RoboDK station: PROYECTO DE MECANIZADO Resuelto.rdk

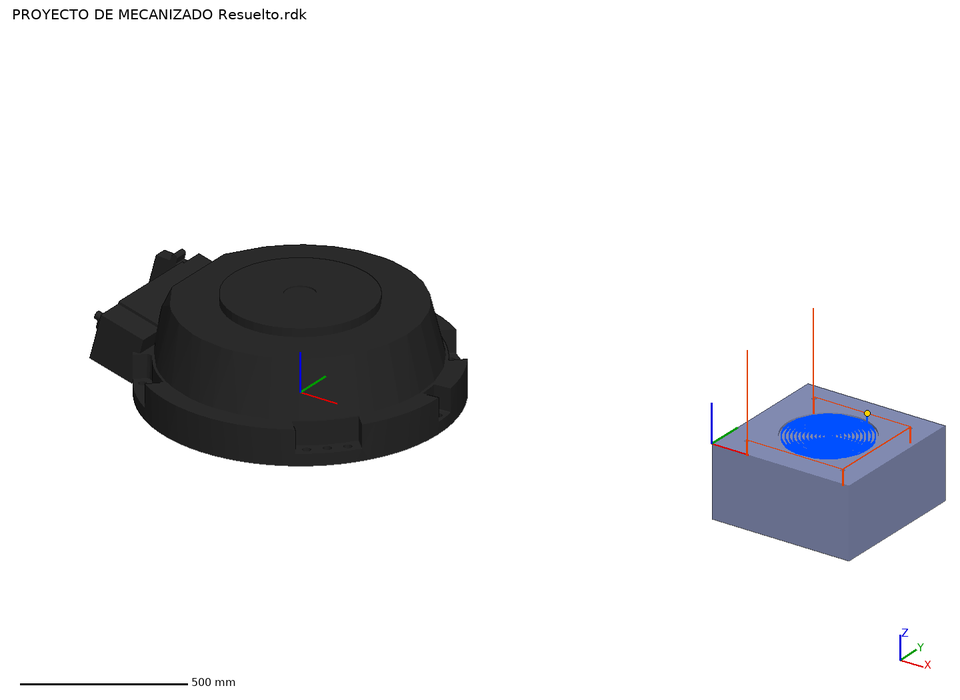
[picture v0: the station drawn from its stored meshes, robots at their saved joint values, targets as dots, program paths as lines]
Station PROYECTO DE MECANIZADO Resuelto (saved by RoboDK 5.7.5). Poses are relative to the parent item; angles as X-Y-Z fixed-axis rotations.
  - frame ORIGEN at (0, 0, 0) mm
  - frame KUKA KR 200 comp Base at (0, 0, 0) mm
    - robot KUKA KR 200 comp: 6 axes
        joint limits [-185, -142, -120, -350, -120, -350] to [185, 0, 148, 350, 120, 350]; home [0, -90, 90, 0, 0, 0]; saved at [-18.305, -63.639, 118.623, 158.005, 56.991, -167.59]
      - tool Teknomotor ATC710039 Spindle, TCP at (296, 0, 80.3) mm, rotated rx 0 ry 90 rz 0 deg, size 475 x 150 x 192.7 mm
        - object ENDMILL_D16_150 at (0, 0, 0) mm, rotated rx 180 ry 0 rz 0 deg, size 16 x 16 x 150 mm, geometry from ENDMILL_D16_150.IGS
  - frame MECANIZADO at (1500, 0, 250) mm
    - object 500x500x250 at (0, 0, 0) mm, size 500 x 500 x 250 mm, geometry from 500x500x250.STEP
  - machining project Machining1 settings: C:/Users/Escritorio/Desktop/pocket_circular (2).gcode | rotZ(0) | rotX(0)*rotY(0)
  - program Machining1 (4843 instructions, listed below)
  - machining project Machining2 settings: C:/Users/Escritorio/Documents/Repos/Proyecto_Tec_12/Proyecto Mecanizado/PROGRAMACION_MANUAL.gcode | rotZ(0) | rotX(0)*rotY(0) | rotz(0) | onStart | onPathStart | onApproach | onPoint | onRetract | onFinish | SetRPM(%1) | SetTool(%1) | Extruder(%1) | default | default | OutOnMov(%1) | OutOffMov(%1) | onPathFinish | M_RunCode(%1)
  - program Machining2 (40 instructions, listed below)
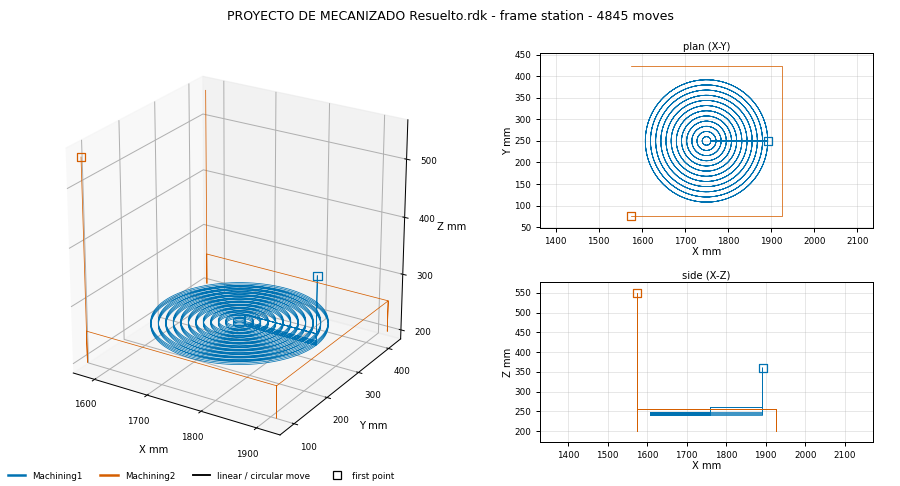
[picture p0: tool path of PROYECTO DE MECANIZADO Resuelto.rdk in frame station, 4845 of 4845 moves have a stored position in this frame; points joined in program order, loops and branches not executed]

--- program Machining1 (robot KUKA KR 200 comp) ---
  Suave(1)
  Establecer velocidad (1000.0 mm/s)
  Est. Ref.: MECANIZADO
  Est. herr: Teknomotor ATC710039 Spindle
  Mostrar Teknomotor ATC710039 Spindle
  MoveJ 1 to (392, 250, 110) mm, rotated rx 180 ry 0 rz -180 deg; joints [-8.871, -45.644, 100.623, 169.209, 55.458, -173.832]
  MoveL 2 to (392, 250, 110) mm, rotated rx 180 ry 0 rz -180 deg; joints [-8.871, -45.644, 100.623, 169.209, 55.458, -173.832]
  MoveL 3 to (392, 250, 10) mm, rotated rx -180 ry 0 rz -180 deg; joints [-8.871, -40.818, 99.818, 169.68, 59.411, -174.706]
  MoveL 4 to (392, 250, 10) mm, rotated rx -180 ry 0 rz -180 deg; joints [-8.871, -40.818, 99.818, 169.68, 59.411, -174.706]
  Establecer velocidad (1000.0 mm/s)
  MoveL 5 to (392, 250, 10) mm, rotated rx -180 ry 0 rz -180 deg; joints [-8.871, -40.818, 99.818, 169.68, 59.411, -174.706]
  Establecer velocidad (1.7 mm/s)
  MoveL 6 to (392, 250, -2.5) mm, rotated rx 180 ry 0 rz 180 deg; joints [-8.871, -40.203, 99.678, 169.73, 59.879, -174.804]
  Establecer velocidad (16.7 mm/s)
  MoveL 7 to (392, 250, -2.5) mm, rotated rx 180 ry 0 rz 180 deg; joints [-8.871, -40.203, 99.678, 169.73, 59.879, -174.804]
  MoveL 8 to (391.71, 259.01, -2.5) mm, rotated rx -180 ry 0 rz -180 deg; joints [-9.187, -40.173, 99.598, 169.361, 59.858, -174.611]
  MoveL 9 to (390.86, 267.98, -2.5) mm, rotated rx -180 ry 0 rz -180 deg; joints [-9.505, -40.157, 99.555, 168.992, 59.862, -174.422]
  MoveL 10 to (389.43, 276.87, -2.5) mm, rotated rx 180 ry 0 rz 180 deg; joints [-9.823, -40.155, 99.548, 168.626, 59.889, -174.237]
  MoveL 11 to (387.45, 285.66, -2.5) mm, rotated rx 180 ry 0 rz 180 deg; joints [-10.141, -40.166, 99.579, 168.263, 59.941, -174.059]
  MoveL 12 to (384.91, 294.31, -2.5) mm, rotated rx 180 ry 0 rz 180 deg; joints [-10.457, -40.191, 99.647, 167.904, 60.016, -173.887]
  MoveL 13 to (381.83, 302.78, -2.5) mm, rotated rx 180 ry 0 rz 180 deg; joints [-10.771, -40.229, 99.751, 167.552, 60.114, -173.723]
  MoveL 14 to (378.22, 311.03, -2.5) mm, rotated rx 180 ry 0 rz -180 deg; joints [-11.082, -40.281, 99.891, 167.207, 60.235, -173.568]
  MoveL 15 to (374.09, 319.04, -2.5) mm, rotated rx -180 ry 0 rz -180 deg; joints [-11.389, -40.346, 100.067, 166.87, 60.378, -173.423]
  MoveL 16 to (369.46, 326.77, -2.5) mm, rotated rx -180 ry 0 rz -180 deg; joints [-11.691, -40.424, 100.278, 166.543, 60.543, -173.289]
  MoveL 17 to (364.35, 334.19, -2.5) mm, rotated rx 180 ry 0 rz 180 deg; joints [-11.987, -40.513, 100.524, 166.226, 60.729, -173.165]
  MoveL 18 to (358.78, 341.28, -2.5) mm, rotated rx -180 ry 0 rz -180 deg; joints [-12.275, -40.615, 100.802, 165.922, 60.935, -173.054]
  MoveL 19 to (352.77, 347.99, -2.5) mm, rotated rx 180 ry 0 rz 180 deg; joints [-12.556, -40.729, 101.113, 165.631, 61.161, -172.955]
  MoveL 20 to (346.35, 354.31, -2.5) mm, rotated rx -180 ry 0 rz 180 deg; joints [-12.828, -40.853, 101.455, 165.353, 61.405, -172.87]
  MoveL 21 to (339.54, 360.21, -2.5) mm, rotated rx -180 ry 0 rz 180 deg; joints [-13.089, -40.987, 101.826, 165.091, 61.667, -172.798]
  MoveL 22 to (332.37, 365.67, -2.5) mm, rotated rx 180 ry 0 rz 180 deg; joints [-13.34, -41.131, 102.226, 164.844, 61.945, -172.74]
  MoveL 23 to (324.87, 370.66, -2.5) mm, rotated rx 180 ry 0 rz 180 deg; joints [-13.579, -41.284, 102.653, 164.614, 62.239, -172.696]
  MoveL 24 to (317.06, 375.17, -2.5) mm, rotated rx -180 ry 0 rz 180 deg; joints [-13.806, -41.445, 103.104, 164.401, 62.548, -172.666]
  MoveL 25 to (308.99, 379.17, -2.5) mm, rotated rx 180 ry 0 rz 180 deg; joints [-14.018, -41.614, 103.579, 164.206, 62.87, -172.65]
  MoveL 26 to (300.68, 382.65, -2.5) mm, rotated rx 180 ry 0 rz -180 deg; joints [-14.217, -41.789, 104.076, 164.03, 63.204, -172.649]
  MoveL 27 to (292.16, 385.6, -2.5) mm, rotated rx 180 ry 0 rz 180 deg; joints [-14.399, -41.97, 104.592, 163.874, 63.55, -172.662]
  MoveL 28 to (283.48, 388, -2.5) mm, rotated rx -180 ry 0 rz 180 deg; joints [-14.566, -42.156, 105.126, 163.737, 63.905, -172.688]
  MoveL 29 to (274.66, 389.84, -2.5) mm, rotated rx 180 ry 0 rz -180 deg; joints [-14.715, -42.347, 105.675, 163.622, 64.269, -172.728]
  MoveL 30 to (265.74, 391.13, -2.5) mm, rotated rx 180 ry 0 rz 180 deg; joints [-14.847, -42.54, 106.238, 163.527, 64.64, -172.782]
  MoveL 31 to (256.76, 391.84, -2.5) mm, rotated rx -180 ry 0 rz 180 deg; joints [-14.96, -42.736, 106.813, 163.454, 65.017, -172.848]
  MoveL 32 to (247.75, 391.98, -2.5) mm, rotated rx -180 ry 0 rz -180 deg; joints [-15.054, -42.934, 107.397, 163.402, 65.399, -172.927]
  MoveL 33 to (238.75, 391.55, -2.5) mm, rotated rx -180 ry 0 rz -180 deg; joints [-15.127, -43.132, 107.987, 163.373, 65.784, -173.017]
  MoveL 34 to (229.79, 390.55, -2.5) mm, rotated rx -180 ry 0 rz -180 deg; joints [-15.18, -43.33, 108.583, 163.367, 66.171, -173.118]
  MoveL 35 to (220.92, 388.99, -2.5) mm, rotated rx -180 ry 0 rz -180 deg; joints [-15.211, -43.526, 109.18, 163.383, 66.559, -173.229]
  MoveL 36 to (212.16, 386.87, -2.5) mm, rotated rx -180 ry 0 rz 180 deg; joints [-15.221, -43.721, 109.778, 163.422, 66.946, -173.351]
  MoveL 37 to (203.56, 384.19, -2.5) mm, rotated rx 180 ry 0 rz -180 deg; joints [-15.208, -43.914, 110.373, 163.484, 67.331, -173.48]
  MoveL 38 to (195.14, 380.97, -2.5) mm, rotated rx 180 ry 0 rz 180 deg; joints [-15.173, -44.102, 110.964, 163.569, 67.712, -173.618]
  MoveL 39 to (186.94, 377.23, -2.5) mm, rotated rx -180 ry 0 rz -180 deg; joints [-15.115, -44.287, 111.547, 163.677, 68.088, -173.763]
  MoveL 40 to (179, 372.98, -2.5) mm, rotated rx -180 ry 0 rz 180 deg; joints [-15.034, -44.466, 112.121, 163.808, 68.458, -173.914]
  MoveL 41 to (171.34, 368.22, -2.5) mm, rotated rx 180 ry 0 rz 180 deg; joints [-14.929, -44.64, 112.683, 163.961, 68.82, -174.07]
  MoveL 42 to (164, 363, -2.5) mm, rotated rx 180 ry 0 rz -180 deg; joints [-14.802, -44.808, 113.231, 164.137, 69.173, -174.231]
  MoveL 43 to (157.01, 357.32, -2.5) mm, rotated rx 180 ry 0 rz -180 deg; joints [-14.652, -44.969, 113.762, 164.335, 69.514, -174.395]
  MoveL 44 to (150.39, 351.2, -2.5) mm, rotated rx 180 ry 0 rz 180 deg; joints [-14.479, -45.122, 114.275, 164.554, 69.844, -174.561]
  MoveL 45 to (144.17, 344.68, -2.5) mm, rotated rx -180 ry 0 rz 180 deg; joints [-14.283, -45.268, 114.767, 164.794, 70.16, -174.729]
  MoveL 46 to (138.38, 337.78, -2.5) mm, rotated rx -180 ry 0 rz 180 deg; joints [-14.067, -45.405, 115.236, 165.054, 70.46, -174.898]
  MoveL 47 to (133.04, 330.52, -2.5) mm, rotated rx 180 ry 0 rz 180 deg; joints [-13.829, -45.533, 115.679, 165.334, 70.744, -175.067]
  MoveL 48 to (128.17, 322.94, -2.5) mm, rotated rx 180 ry 0 rz 180 deg; joints [-13.571, -45.653, 116.096, 165.632, 71.01, -175.235]
  MoveL 49 to (123.79, 315.07, -2.5) mm, rotated rx 180 ry 0 rz -180 deg; joints [-13.294, -45.763, 116.484, 165.947, 71.257, -175.402]
  MoveL 50 to (119.91, 306.93, -2.5) mm, rotated rx -180 ry 0 rz -180 deg; joints [-12.999, -45.863, 116.841, 166.278, 71.484, -175.566]
  MoveL 51 to (116.56, 298.57, -2.5) mm, rotated rx -180 ry 0 rz -180 deg; joints [-12.687, -45.953, 117.166, 166.624, 71.688, -175.727]
  MoveL 52 to (113.75, 290.01, -2.5) mm, rotated rx 180 ry 0 rz 180 deg; joints [-12.36, -46.034, 117.458, 166.983, 71.87, -175.885]
  MoveL 53 to (111.49, 281.28, -2.5) mm, rotated rx 180 ry 0 rz -180 deg; joints [-12.019, -46.104, 117.714, 167.355, 72.027, -176.04]
  MoveL 54 to (109.78, 272.44, -2.5) mm, rotated rx -180 ry 0 rz 180 deg; joints [-11.666, -46.164, 117.934, 167.736, 72.16, -176.19]
  MoveL 55 to (108.64, 263.5, -2.5) mm, rotated rx 180 ry 0 rz -180 deg; joints [-11.303, -46.213, 118.117, 168.125, 72.267, -176.335]
  MoveL 56 to (108.07, 254.51, -2.5) mm, rotated rx -180 ry 0 rz 180 deg; joints [-10.931, -46.252, 118.261, 168.522, 72.347, -176.476]
  MoveL 57 to (108.07, 245.49, -2.5) mm, rotated rx 180 ry 0 rz -180 deg; joints [-10.553, -46.28, 118.367, 168.922, 72.4, -176.612]
  MoveL 58 to (108.64, 236.5, -2.5) mm, rotated rx 180 ry 0 rz -180 deg; joints [-10.17, -46.298, 118.434, 169.326, 72.426, -176.743]
  MoveL 59 to (109.78, 227.56, -2.5) mm, rotated rx -180 ry 0 rz 180 deg; joints [-9.785, -46.305, 118.46, 169.731, 72.423, -176.868]
  MoveL 60 to (111.49, 218.72, -2.5) mm, rotated rx -180 ry 0 rz -180 deg; joints [-9.4, -46.302, 118.447, 170.134, 72.393, -176.989]
  MoveL 61 to (113.75, 209.99, -2.5) mm, rotated rx -180 ry 0 rz -180 deg; joints [-9.016, -46.288, 118.395, 170.534, 72.335, -177.104]
  MoveL 62 to (116.56, 201.43, -2.5) mm, rotated rx 180 ry 0 rz -180 deg; joints [-8.636, -46.263, 118.302, 170.929, 72.25, -177.213]
  MoveL 63 to (119.91, 193.07, -2.5) mm, rotated rx -180 ry 0 rz 180 deg; joints [-8.262, -46.228, 118.171, 171.316, 72.137, -177.318]
  MoveL 64 to (123.79, 184.93, -2.5) mm, rotated rx 180 ry 0 rz -180 deg; joints [-7.896, -46.182, 118.001, 171.695, 71.998, -177.417]
  MoveL 65 to (128.17, 177.06, -2.5) mm, rotated rx -180 ry 0 rz 180 deg; joints [-7.539, -46.126, 117.794, 172.063, 71.832, -177.511]
  MoveL 66 to (133.04, 169.48, -2.5) mm, rotated rx 180 ry 0 rz 180 deg; joints [-7.194, -46.059, 117.55, 172.418, 71.642, -177.599]
  MoveL 67 to (138.38, 162.22, -2.5) mm, rotated rx 180 ry 0 rz -180 deg; joints [-6.862, -45.982, 117.271, 172.759, 71.427, -177.683]
  MoveL 68 to (144.17, 155.32, -2.5) mm, rotated rx -180 ry 0 rz -180 deg; joints [-6.544, -45.895, 116.957, 173.085, 71.19, -177.76]
  MoveL 69 to (150.39, 148.8, -2.5) mm, rotated rx 180 ry 0 rz -180 deg; joints [-6.243, -45.799, 116.611, 173.392, 70.931, -177.833]
  MoveL 70 to (157.01, 142.68, -2.5) mm, rotated rx 180 ry 0 rz -180 deg; joints [-5.96, -45.692, 116.233, 173.682, 70.651, -177.899]
  MoveL 71 to (164, 137, -2.5) mm, rotated rx -180 ry 0 rz 180 deg; joints [-5.695, -45.576, 115.826, 173.951, 70.352, -177.959]
  MoveL 72 to (171.34, 131.78, -2.5) mm, rotated rx 180 ry 0 rz -180 deg; joints [-5.45, -45.45, 115.392, 174.2, 70.036, -178.014]
  MoveL 73 to (179, 127.02, -2.5) mm, rotated rx 180 ry 0 rz 180 deg; joints [-5.226, -45.316, 114.931, 174.427, 69.704, -178.061]
  MoveL 74 to (186.94, 122.77, -2.5) mm, rotated rx -180 ry 0 rz 180 deg; joints [-5.024, -45.174, 114.447, 174.631, 69.357, -178.102]
  MoveL 75 to (195.14, 119.03, -2.5) mm, rotated rx 180 ry 0 rz 180 deg; joints [-4.843, -45.023, 113.941, 174.812, 68.997, -178.136]
  MoveL 76 to (203.56, 115.81, -2.5) mm, rotated rx 180 ry 0 rz 180 deg; joints [-4.685, -44.864, 113.416, 174.969, 68.627, -178.162]
  MoveL 77 to (212.16, 113.13, -2.5) mm, rotated rx 180 ry 0 rz -180 deg; joints [-4.549, -44.699, 112.874, 175.101, 68.247, -178.181]
  MoveL 78 to (220.92, 111.01, -2.5) mm, rotated rx -180 ry 0 rz 180 deg; joints [-4.437, -44.527, 112.316, 175.209, 67.859, -178.191]
  MoveL 79 to (229.79, 109.45, -2.5) mm, rotated rx -180 ry 0 rz -180 deg; joints [-4.348, -44.349, 111.746, 175.292, 67.466, -178.192]
  MoveL 80 to (238.75, 108.45, -2.5) mm, rotated rx -180 ry 0 rz 180 deg; joints [-4.282, -44.167, 111.166, 175.35, 67.067, -178.185]
  MoveL 81 to (247.75, 108.02, -2.5) mm, rotated rx -180 ry 0 rz -180 deg; joints [-4.239, -43.979, 110.578, 175.383, 66.666, -178.168]
  MoveL 82 to (256.76, 108.16, -2.5) mm, rotated rx -180 ry 0 rz -180 deg; joints [-4.218, -43.788, 109.984, 175.391, 66.264, -178.141]
  MoveL 83 to (265.74, 108.87, -2.5) mm, rotated rx 180 ry 0 rz 180 deg; joints [-4.22, -43.594, 109.387, 175.375, 65.863, -178.105]
  MoveL 84 to (274.66, 110.16, -2.5) mm, rotated rx 180 ry 0 rz 180 deg; joints [-4.244, -43.398, 108.789, 175.334, 65.463, -178.059]
  MoveL 85 to (283.48, 112, -2.5) mm, rotated rx 180 ry 0 rz 180 deg; joints [-4.29, -43.2, 108.193, 175.268, 65.067, -178.002]
  MoveL 86 to (292.16, 114.4, -2.5) mm, rotated rx -180 ry 0 rz 180 deg; joints [-4.356, -43.002, 107.6, 175.18, 64.677, -177.934]
  MoveL 87 to (300.68, 117.35, -2.5) mm, rotated rx -180 ry 0 rz -180 deg; joints [-4.443, -42.804, 107.014, 175.068, 64.293, -177.856]
  MoveL 88 to (308.99, 120.83, -2.5) mm, rotated rx 180 ry 0 rz 180 deg; joints [-4.549, -42.608, 106.436, 174.934, 63.917, -177.768]
  MoveL 89 to (317.06, 124.83, -2.5) mm, rotated rx -180 ry 0 rz -180 deg; joints [-4.674, -42.413, 105.868, 174.778, 63.55, -177.669]
  MoveL 90 to (324.87, 129.34, -2.5) mm, rotated rx -180 ry 0 rz -180 deg; joints [-4.818, -42.222, 105.314, 174.601, 63.195, -177.559]
  MoveL 91 to (332.37, 134.33, -2.5) mm, rotated rx -180 ry 0 rz 180 deg; joints [-4.978, -42.034, 104.774, 174.403, 62.852, -177.44]
  MoveL 92 to (339.54, 139.79, -2.5) mm, rotated rx -180 ry 0 rz -180 deg; joints [-5.156, -41.851, 104.252, 174.186, 62.522, -177.31]
  MoveL 93 to (346.35, 145.69, -2.5) mm, rotated rx -180 ry 0 rz -180 deg; joints [-5.349, -41.674, 103.748, 173.951, 62.207, -177.171]
  MoveL 94 to (352.77, 152.01, -2.5) mm, rotated rx -180 ry 0 rz 180 deg; joints [-5.557, -41.503, 103.266, 173.698, 61.907, -177.023]
  MoveL 95 to (358.78, 158.72, -2.5) mm, rotated rx -180 ry 0 rz -180 deg; joints [-5.778, -41.339, 102.806, 173.429, 61.625, -176.867]
  MoveL 96 to (364.35, 165.81, -2.5) mm, rotated rx 180 ry 0 rz 180 deg; joints [-6.013, -41.183, 102.37, 173.145, 61.361, -176.702]
  MoveL 97 to (369.46, 173.23, -2.5) mm, rotated rx 180 ry 0 rz 180 deg; joints [-6.26, -41.036, 101.961, 172.846, 61.115, -176.53]
  MoveL 98 to (374.09, 180.96, -2.5) mm, rotated rx 180 ry 0 rz -180 deg; joints [-6.518, -40.898, 101.58, 172.534, 60.89, -176.352]
  MoveL 99 to (378.22, 188.97, -2.5) mm, rotated rx 180 ry 0 rz 180 deg; joints [-6.787, -40.77, 101.228, 172.211, 60.685, -176.168]
  MoveL 100 to (381.83, 197.22, -2.5) mm, rotated rx 180 ry 0 rz 180 deg; joints [-7.064, -40.653, 100.906, 171.877, 60.501, -175.98]
  MoveL 101 to (384.91, 205.69, -2.5) mm, rotated rx 180 ry 0 rz 180 deg; joints [-7.35, -40.547, 100.616, 171.534, 60.34, -175.787]
  MoveL 102 to (387.45, 214.34, -2.5) mm, rotated rx -180 ry 0 rz 180 deg; joints [-7.643, -40.453, 100.359, 171.183, 60.201, -175.592]
  MoveL 103 to (389.43, 223.13, -2.5) mm, rotated rx 180 ry 0 rz 180 deg; joints [-7.943, -40.371, 100.136, 170.826, 60.085, -175.395]
  MoveL 104 to (390.86, 232.02, -2.5) mm, rotated rx -180 ry 0 rz -180 deg; joints [-8.248, -40.302, 99.948, 170.464, 59.992, -175.198]
  MoveL 105 to (391.71, 240.99, -2.5) mm, rotated rx 180 ry 0 rz 180 deg; joints [-8.558, -40.246, 99.795, 170.098, 59.924, -175]
  MoveL 106 to (392, 250, -2.5) mm, rotated rx 180 ry 0 rz 180 deg; joints [-8.871, -40.203, 99.678, 169.73, 59.879, -174.804]
  MoveL 107 to (380, 250, -2.5) mm, rotated rx -180 ry 0 rz -180 deg; joints [-8.937, -40.511, 100.517, 169.708, 60.406, -174.876]
  MoveL 108 to (379.74, 258.25, -2.5) mm, rotated rx 180 ry 0 rz 180 deg; joints [-9.229, -40.484, 100.443, 169.37, 60.387, -174.701]
  MoveL 109 to (378.95, 266.46, -2.5) mm, rotated rx 180 ry 0 rz -180 deg; joints [-9.521, -40.469, 100.403, 169.032, 60.39, -174.53]
  MoveL 110 to (377.65, 274.6, -2.5) mm, rotated rx 180 ry 0 rz 180 deg; joints [-9.815, -40.467, 100.397, 168.696, 60.415, -174.364]
  MoveL 111 to (375.83, 282.65, -2.5) mm, rotated rx -180 ry 0 rz -180 deg; joints [-10.108, -40.477, 100.425, 168.362, 60.461, -174.202]
  MoveL 112 to (373.51, 290.56, -2.5) mm, rotated rx 180 ry 0 rz -180 deg; joints [-10.4, -40.5, 100.487, 168.033, 60.529, -174.047]
  MoveL 113 to (370.69, 298.32, -2.5) mm, rotated rx -180 ry 0 rz -180 deg; joints [-10.689, -40.535, 100.583, 167.71, 60.619, -173.899]
  MoveL 114 to (367.38, 305.87, -2.5) mm, rotated rx -180 ry 0 rz 180 deg; joints [-10.976, -40.582, 100.712, 167.393, 60.73, -173.759]
  MoveL 115 to (363.6, 313.21, -2.5) mm, rotated rx -180 ry 0 rz -180 deg; joints [-11.259, -40.641, 100.873, 167.083, 60.861, -173.628]
  MoveL 116 to (359.36, 320.28, -2.5) mm, rotated rx 180 ry 0 rz -180 deg; joints [-11.537, -40.712, 101.067, 166.783, 61.012, -173.506]
  MoveL 117 to (354.69, 327.08, -2.5) mm, rotated rx 180 ry 0 rz 180 deg; joints [-11.809, -40.793, 101.291, 166.492, 61.182, -173.395]
  MoveL 118 to (349.59, 333.56, -2.5) mm, rotated rx 180 ry 0 rz -180 deg; joints [-12.075, -40.886, 101.547, 166.212, 61.371, -173.294]
  MoveL 119 to (344.09, 339.71, -2.5) mm, rotated rx -180 ry 0 rz 180 deg; joints [-12.333, -40.989, 101.832, 165.944, 61.578, -173.205]
  MoveL 120 to (338.21, 345.5, -2.5) mm, rotated rx -180 ry 0 rz -180 deg; joints [-12.582, -41.102, 102.145, 165.689, 61.802, -173.127]
  MoveL 121 to (331.97, 350.9, -2.5) mm, rotated rx 180 ry 0 rz 180 deg; joints [-12.823, -41.224, 102.486, 165.448, 62.042, -173.061]
  MoveL 122 to (325.41, 355.89, -2.5) mm, rotated rx 180 ry 0 rz 180 deg; joints [-13.053, -41.355, 102.852, 165.221, 62.298, -173.008]
  MoveL 123 to (318.54, 360.46, -2.5) mm, rotated rx 180 ry 0 rz 180 deg; joints [-13.272, -41.495, 103.243, 165.01, 62.567, -172.967]
  MoveL 124 to (311.4, 364.59, -2.5) mm, rotated rx 180 ry 0 rz 180 deg; joints [-13.479, -41.641, 103.657, 164.814, 62.851, -172.94]
  MoveL 125 to (304, 368.25, -2.5) mm, rotated rx 180 ry 0 rz 180 deg; joints [-13.673, -41.795, 104.092, 164.636, 63.147, -172.925]
  MoveL 126 to (296.4, 371.44, -2.5) mm, rotated rx -180 ry 0 rz 180 deg; joints [-13.854, -41.955, 104.547, 164.474, 63.454, -172.922]
  MoveL 127 to (288.6, 374.14, -2.5) mm, rotated rx 180 ry 0 rz 180 deg; joints [-14.02, -42.12, 105.02, 164.331, 63.771, -172.933]
  MoveL 128 to (280.65, 376.34, -2.5) mm, rotated rx 180 ry 0 rz -180 deg; joints [-14.172, -42.29, 105.51, 164.206, 64.097, -172.956]
  MoveL 129 to (272.57, 378.03, -2.5) mm, rotated rx 180 ry 0 rz -180 deg; joints [-14.307, -42.463, 106.013, 164.101, 64.431, -172.991]
  MoveL 130 to (264.41, 379.2, -2.5) mm, rotated rx -180 ry 0 rz -180 deg; joints [-14.426, -42.64, 106.53, 164.014, 64.772, -173.039]
  MoveL 131 to (256.19, 379.85, -2.5) mm, rotated rx -180 ry 0 rz 180 deg; joints [-14.527, -42.818, 107.056, 163.948, 65.118, -173.097]
  MoveL 132 to (247.94, 379.98, -2.5) mm, rotated rx 180 ry 0 rz 180 deg; joints [-14.611, -42.999, 107.591, 163.902, 65.469, -173.167]
  MoveL 133 to (239.7, 379.59, -2.5) mm, rotated rx 180 ry 0 rz -180 deg; joints [-14.676, -43.18, 108.132, 163.876, 65.822, -173.248]
  MoveL 134 to (231.5, 378.68, -2.5) mm, rotated rx -180 ry 0 rz 180 deg; joints [-14.722, -43.361, 108.677, 163.872, 66.178, -173.338]
  MoveL 135 to (223.38, 377.24, -2.5) mm, rotated rx 180 ry 0 rz 180 deg; joints [-14.748, -43.541, 109.224, 163.888, 66.534, -173.438]
  MoveL 136 to (215.36, 375.3, -2.5) mm, rotated rx 180 ry 0 rz -180 deg; joints [-14.754, -43.719, 109.771, 163.925, 66.889, -173.547]
  MoveL 137 to (207.48, 372.85, -2.5) mm, rotated rx -180 ry 0 rz 180 deg; joints [-14.74, -43.895, 110.316, 163.983, 67.241, -173.663]
  MoveL 138 to (199.78, 369.91, -2.5) mm, rotated rx 180 ry 0 rz -180 deg; joints [-14.705, -44.068, 110.857, 164.063, 67.591, -173.787]
  MoveL 139 to (192.27, 366.48, -2.5) mm, rotated rx 180 ry 0 rz 180 deg; joints [-14.649, -44.238, 111.391, 164.164, 67.935, -173.918]
  MoveL 140 to (185, 362.58, -2.5) mm, rotated rx 180 ry 0 rz 180 deg; joints [-14.573, -44.402, 111.915, 164.285, 68.274, -174.054]
  MoveL 141 to (177.99, 358.23, -2.5) mm, rotated rx 180 ry 0 rz 180 deg; joints [-14.475, -44.562, 112.429, 164.428, 68.605, -174.195]
  MoveL 142 to (171.27, 353.45, -2.5) mm, rotated rx -180 ry 0 rz 180 deg; joints [-14.356, -44.716, 112.93, 164.59, 68.927, -174.34]
  MoveL 143 to (164.87, 348.25, -2.5) mm, rotated rx 180 ry 0 rz -180 deg; joints [-14.217, -44.864, 113.416, 164.773, 69.239, -174.489]
  MoveL 144 to (158.81, 342.65, -2.5) mm, rotated rx 180 ry 0 rz -180 deg; joints [-14.057, -45.006, 113.885, 164.975, 69.54, -174.64]
  MoveL 145 to (153.12, 336.68, -2.5) mm, rotated rx 180 ry 0 rz 180 deg; joints [-13.877, -45.14, 114.334, 165.196, 69.828, -174.793]
  MoveL 146 to (147.81, 330.36, -2.5) mm, rotated rx -180 ry 0 rz 180 deg; joints [-13.677, -45.266, 114.762, 165.436, 70.102, -174.947]
  MoveL 147 to (142.92, 323.72, -2.5) mm, rotated rx 180 ry 0 rz -180 deg; joints [-13.459, -45.385, 115.167, 165.692, 70.36, -175.101]
  MoveL 148 to (138.46, 316.78, -2.5) mm, rotated rx 180 ry 0 rz 180 deg; joints [-13.223, -45.496, 115.548, 165.966, 70.602, -175.254]
  MoveL 149 to (134.45, 309.57, -2.5) mm, rotated rx -180 ry 0 rz -180 deg; joints [-12.97, -45.597, 115.902, 166.254, 70.827, -175.407]
  MoveL 150 to (130.91, 302.12, -2.5) mm, rotated rx 180 ry 0 rz 180 deg; joints [-12.7, -45.69, 116.228, 166.557, 71.032, -175.558]
  MoveL 151 to (127.84, 294.46, -2.5) mm, rotated rx 180 ry 0 rz 180 deg; joints [-12.416, -45.774, 116.524, 166.874, 71.217, -175.706]
  MoveL 152 to (125.27, 286.63, -2.5) mm, rotated rx -180 ry 0 rz -180 deg; joints [-12.118, -45.849, 116.79, 167.202, 71.382, -175.852]
  MoveL 153 to (123.19, 278.64, -2.5) mm, rotated rx 180 ry 0 rz 180 deg; joints [-11.808, -45.914, 117.024, 167.541, 71.524, -175.995]
  MoveL 154 to (121.63, 270.54, -2.5) mm, rotated rx 180 ry 0 rz 180 deg; joints [-11.487, -45.969, 117.224, 167.888, 71.644, -176.134]
  MoveL 155 to (120.59, 262.36, -2.5) mm, rotated rx 180 ry 0 rz 180 deg; joints [-11.157, -46.015, 117.391, 168.244, 71.74, -176.269]
  MoveL 156 to (120.07, 254.12, -2.5) mm, rotated rx 180 ry 0 rz 180 deg; joints [-10.819, -46.052, 117.522, 168.605, 71.812, -176.4]
  MoveL 157 to (120.07, 245.88, -2.5) mm, rotated rx -180 ry 0 rz -180 deg; joints [-10.476, -46.078, 117.619, 168.97, 71.859, -176.527]
  MoveL 158 to (120.59, 237.64, -2.5) mm, rotated rx -180 ry 0 rz -180 deg; joints [-10.128, -46.094, 117.679, 169.337, 71.882, -176.649]
  MoveL 159 to (121.63, 229.46, -2.5) mm, rotated rx 180 ry 0 rz 180 deg; joints [-9.779, -46.101, 117.704, 169.705, 71.879, -176.767]
  MoveL 160 to (123.19, 221.36, -2.5) mm, rotated rx 180 ry 0 rz 180 deg; joints [-9.429, -46.098, 117.692, 170.072, 71.851, -176.879]
  MoveL 161 to (125.27, 213.37, -2.5) mm, rotated rx 180 ry 0 rz 180 deg; joints [-9.081, -46.085, 117.644, 170.436, 71.798, -176.987]
  MoveL 162 to (127.84, 205.54, -2.5) mm, rotated rx -180 ry 0 rz 180 deg; joints [-8.736, -46.062, 117.56, 170.796, 71.72, -177.09]
  MoveL 163 to (130.91, 197.88, -2.5) mm, rotated rx 180 ry 0 rz 180 deg; joints [-8.396, -46.029, 117.44, 171.149, 71.618, -177.188]
  MoveL 164 to (134.45, 190.43, -2.5) mm, rotated rx 180 ry 0 rz -180 deg; joints [-8.064, -45.986, 117.286, 171.493, 71.491, -177.282]
  MoveL 165 to (138.46, 183.22, -2.5) mm, rotated rx 180 ry 0 rz 180 deg; joints [-7.739, -45.934, 117.097, 171.828, 71.34, -177.37]
  MoveL 166 to (142.92, 176.28, -2.5) mm, rotated rx -180 ry 0 rz 180 deg; joints [-7.425, -45.872, 116.874, 172.152, 71.167, -177.452]
  MoveL 167 to (147.81, 169.64, -2.5) mm, rotated rx 180 ry 0 rz 180 deg; joints [-7.123, -45.801, 116.619, 172.463, 70.972, -177.53]
  MoveL 168 to (153.12, 163.32, -2.5) mm, rotated rx -180 ry 0 rz 180 deg; joints [-6.834, -45.72, 116.333, 172.76, 70.756, -177.602]
  MoveL 169 to (158.81, 157.35, -2.5) mm, rotated rx 180 ry 0 rz 180 deg; joints [-6.559, -45.63, 116.017, 173.041, 70.521, -177.669]
  MoveL 170 to (164.87, 151.75, -2.5) mm, rotated rx 180 ry 0 rz -180 deg; joints [-6.3, -45.532, 115.673, 173.305, 70.266, -177.73]
  MoveL 171 to (171.27, 146.55, -2.5) mm, rotated rx -180 ry 0 rz 180 deg; joints [-6.058, -45.424, 115.301, 173.552, 69.994, -177.786]
  MoveL 172 to (177.99, 141.77, -2.5) mm, rotated rx 180 ry 0 rz -180 deg; joints [-5.833, -45.308, 114.905, 173.779, 69.707, -177.835]
  MoveL 173 to (185, 137.42, -2.5) mm, rotated rx -180 ry 0 rz 180 deg; joints [-5.627, -45.184, 114.484, 173.987, 69.404, -177.878]
  MoveL 174 to (192.27, 133.52, -2.5) mm, rotated rx 180 ry 0 rz -180 deg; joints [-5.44, -45.053, 114.042, 174.175, 69.088, -177.915]
  MoveL 175 to (199.78, 130.09, -2.5) mm, rotated rx 180 ry 0 rz 180 deg; joints [-5.273, -44.914, 113.58, 174.341, 68.761, -177.944]
  MoveL 176 to (207.48, 127.15, -2.5) mm, rotated rx 180 ry 0 rz -180 deg; joints [-5.127, -44.768, 113.1, 174.486, 68.423, -177.967]
  MoveL 177 to (215.36, 124.7, -2.5) mm, rotated rx -180 ry 0 rz 180 deg; joints [-5.001, -44.616, 112.604, 174.608, 68.076, -177.982]
  MoveL 178 to (223.38, 122.76, -2.5) mm, rotated rx -180 ry 0 rz -180 deg; joints [-4.896, -44.458, 112.094, 174.708, 67.722, -177.989]
  MoveL 179 to (231.5, 121.32, -2.5) mm, rotated rx 180 ry 0 rz 180 deg; joints [-4.812, -44.295, 111.573, 174.785, 67.362, -177.988]
  MoveL 180 to (239.7, 120.41, -2.5) mm, rotated rx 180 ry 0 rz 180 deg; joints [-4.749, -44.127, 111.042, 174.84, 66.998, -177.979]
  MoveL 181 to (247.94, 120.02, -2.5) mm, rotated rx 180 ry 0 rz -180 deg; joints [-4.707, -43.955, 110.504, 174.871, 66.632, -177.961]
  MoveL 182 to (256.19, 120.15, -2.5) mm, rotated rx 180 ry 0 rz -180 deg; joints [-4.686, -43.78, 109.96, 174.88, 66.264, -177.935]
  MoveL 183 to (264.41, 120.8, -2.5) mm, rotated rx 180 ry 0 rz 180 deg; joints [-4.685, -43.603, 109.413, 174.867, 65.897, -177.899]
  MoveL 184 to (272.57, 121.98, -2.5) mm, rotated rx -180 ry 0 rz -180 deg; joints [-4.704, -43.423, 108.866, 174.83, 65.531, -177.854]
  MoveL 185 to (280.65, 123.66, -2.5) mm, rotated rx -180 ry 0 rz -180 deg; joints [-4.743, -43.242, 108.32, 174.772, 65.168, -177.8]
  MoveL 186 to (288.6, 125.86, -2.5) mm, rotated rx 180 ry 0 rz 180 deg; joints [-4.802, -43.061, 107.777, 174.692, 64.811, -177.736]
  MoveL 187 to (296.4, 128.56, -2.5) mm, rotated rx -180 ry 0 rz 180 deg; joints [-4.879, -42.881, 107.24, 174.591, 64.459, -177.662]
  MoveL 188 to (304, 131.75, -2.5) mm, rotated rx 180 ry 0 rz -180 deg; joints [-4.974, -42.701, 106.71, 174.469, 64.114, -177.579]
  MoveL 189 to (311.4, 135.41, -2.5) mm, rotated rx 180 ry 0 rz 180 deg; joints [-5.087, -42.524, 106.19, 174.327, 63.778, -177.487]
  MoveL 190 to (318.54, 139.54, -2.5) mm, rotated rx 180 ry 0 rz -180 deg; joints [-5.217, -42.349, 105.682, 174.166, 63.452, -177.385]
  MoveL 191 to (325.41, 144.11, -2.5) mm, rotated rx 180 ry 0 rz -180 deg; joints [-5.363, -42.178, 105.188, 173.986, 63.137, -177.275]
  MoveL 192 to (331.97, 149.1, -2.5) mm, rotated rx -180 ry 0 rz 180 deg; joints [-5.524, -42.011, 104.709, 173.788, 62.835, -177.155]
  MoveL 193 to (338.21, 154.5, -2.5) mm, rotated rx 180 ry 0 rz 180 deg; joints [-5.7, -41.849, 104.247, 173.574, 62.546, -177.027]
  MoveL 194 to (344.09, 160.29, -2.5) mm, rotated rx 180 ry 0 rz -180 deg; joints [-5.89, -41.694, 103.805, 173.343, 62.271, -176.891]
  MoveL 195 to (349.59, 166.44, -2.5) mm, rotated rx 180 ry 0 rz 180 deg; joints [-6.093, -41.544, 103.383, 173.097, 62.012, -176.748]
  MoveL 196 to (354.69, 172.92, -2.5) mm, rotated rx -180 ry 0 rz 180 deg; joints [-6.308, -41.403, 102.984, 172.837, 61.769, -176.598]
  MoveL 197 to (359.36, 179.72, -2.5) mm, rotated rx 180 ry 0 rz -180 deg; joints [-6.534, -41.269, 102.609, 172.563, 61.544, -176.441]
  MoveL 198 to (363.6, 186.79, -2.5) mm, rotated rx -180 ry 0 rz -180 deg; joints [-6.771, -41.143, 102.26, 172.278, 61.337, -176.279]
  MoveL 199 to (367.38, 194.13, -2.5) mm, rotated rx -180 ry 0 rz 180 deg; joints [-7.017, -41.027, 101.937, 171.982, 61.148, -176.111]
  MoveL 200 to (370.69, 201.68, -2.5) mm, rotated rx -180 ry 0 rz 180 deg; joints [-7.273, -40.92, 101.642, 171.676, 60.98, -175.94]
  MoveL 201 to (373.51, 209.44, -2.5) mm, rotated rx 180 ry 0 rz -180 deg; joints [-7.536, -40.824, 101.376, 171.362, 60.831, -175.766]
  MoveL 202 to (375.83, 217.35, -2.5) mm, rotated rx 180 ry 0 rz -180 deg; joints [-7.806, -40.739, 101.141, 171.041, 60.703, -175.589]
  MoveL 203 to (377.65, 225.4, -2.5) mm, rotated rx 180 ry 0 rz -180 deg; joints [-8.082, -40.664, 100.936, 170.713, 60.597, -175.41]
  MoveL 204 to (378.95, 233.54, -2.5) mm, rotated rx 180 ry 0 rz 180 deg; joints [-8.363, -40.601, 100.764, 170.381, 60.511, -175.231]
  MoveL 205 to (379.74, 241.75, -2.5) mm, rotated rx 180 ry 0 rz 180 deg; joints [-8.648, -40.55, 100.624, 170.046, 60.448, -175.053]
  MoveL 206 to (380, 250, -2.5) mm, rotated rx -180 ry 0 rz -180 deg; joints [-8.937, -40.511, 100.517, 169.708, 60.406, -174.876]
  MoveL 207 to (368, 250, -2.5) mm, rotated rx -180 ry 0 rz -180 deg; joints [-9.004, -40.814, 101.349, 169.685, 60.933, -174.947]
  MoveL 208 to (367.76, 257.48, -2.5) mm, rotated rx 180 ry 0 rz -180 deg; joints [-9.27, -40.79, 101.283, 169.377, 60.915, -174.791]
  MoveL 209 to (367.05, 264.94, -2.5) mm, rotated rx -180 ry 0 rz -180 deg; joints [-9.538, -40.777, 101.246, 169.07, 60.917, -174.637]
  MoveL 210 to (365.87, 272.33, -2.5) mm, rotated rx 180 ry 0 rz -180 deg; joints [-9.806, -40.775, 101.241, 168.764, 60.939, -174.488]
  MoveL 211 to (364.22, 279.64, -2.5) mm, rotated rx -180 ry 0 rz -180 deg; joints [-10.075, -40.784, 101.267, 168.461, 60.981, -174.344]
  MoveL 212 to (362.11, 286.82, -2.5) mm, rotated rx -180 ry 0 rz 180 deg; joints [-10.341, -40.805, 101.323, 168.161, 61.043, -174.205]
  MoveL 213 to (359.55, 293.86, -2.5) mm, rotated rx 180 ry 0 rz 180 deg; joints [-10.606, -40.836, 101.41, 167.866, 61.124, -174.072]
  MoveL 214 to (356.55, 300.72, -2.5) mm, rotated rx 180 ry 0 rz 180 deg; joints [-10.868, -40.879, 101.527, 167.578, 61.224, -173.947]
  MoveL 215 to (353.11, 307.37, -2.5) mm, rotated rx -180 ry 0 rz 180 deg; joints [-11.127, -40.932, 101.673, 167.296, 61.343, -173.83]
  MoveL 216 to (349.27, 313.8, -2.5) mm, rotated rx -180 ry 0 rz -180 deg; joints [-11.381, -40.995, 101.849, 167.022, 61.48, -173.721]
  MoveL 217 to (345.02, 319.96, -2.5) mm, rotated rx -180 ry 0 rz -180 deg; joints [-11.629, -41.069, 102.054, 166.757, 61.635, -173.62]
  MoveL 218 to (340.39, 325.85, -2.5) mm, rotated rx -180 ry 0 rz -180 deg; joints [-11.871, -41.153, 102.286, 166.502, 61.807, -173.53]
  MoveL 219 to (335.4, 331.43, -2.5) mm, rotated rx -180 ry 0 rz -180 deg; joints [-12.107, -41.246, 102.545, 166.258, 61.995, -173.45]
  MoveL 220 to (330.06, 336.68, -2.5) mm, rotated rx -180 ry 0 rz -180 deg; joints [-12.334, -41.347, 102.83, 166.026, 62.198, -173.379]
  MoveL 221 to (324.41, 341.59, -2.5) mm, rotated rx -180 ry 0 rz -180 deg; joints [-12.553, -41.458, 103.139, 165.806, 62.417, -173.32]
  MoveL 222 to (318.45, 346.12, -2.5) mm, rotated rx 180 ry 0 rz 180 deg; joints [-12.762, -41.576, 103.472, 165.599, 62.65, -173.272]
  MoveL 223 to (312.21, 350.27, -2.5) mm, rotated rx -180 ry 0 rz 180 deg; joints [-12.961, -41.702, 103.828, 165.407, 62.895, -173.235]
  MoveL 224 to (305.73, 354.01, -2.5) mm, rotated rx -180 ry 0 rz 180 deg; joints [-13.149, -41.834, 104.204, 165.229, 63.153, -173.209]
  MoveL 225 to (299.02, 357.34, -2.5) mm, rotated rx -180 ry 0 rz -180 deg; joints [-13.325, -41.973, 104.6, 165.066, 63.422, -173.195]
  MoveL 226 to (292.11, 360.23, -2.5) mm, rotated rx -180 ry 0 rz -180 deg; joints [-13.488, -42.117, 105.013, 164.92, 63.702, -173.192]
  MoveL 227 to (285.04, 362.68, -2.5) mm, rotated rx 180 ry 0 rz -180 deg; joints [-13.639, -42.266, 105.443, 164.789, 63.991, -173.201]
  MoveL 228 to (277.82, 364.67, -2.5) mm, rotated rx 180 ry 0 rz 180 deg; joints [-13.775, -42.42, 105.888, 164.676, 64.288, -173.22]
  MoveL 229 to (270.49, 366.21, -2.5) mm, rotated rx -180 ry 0 rz 180 deg; joints [-13.896, -42.577, 106.346, 164.581, 64.592, -173.251]
  MoveL 230 to (263.08, 367.27, -2.5) mm, rotated rx -180 ry 0 rz -180 deg; joints [-14.002, -42.737, 106.814, 164.503, 64.903, -173.292]
  MoveL 231 to (255.61, 367.87, -2.5) mm, rotated rx -180 ry 0 rz 180 deg; joints [-14.093, -42.898, 107.293, 164.443, 65.218, -173.344]
  MoveL 232 to (248.13, 367.99, -2.5) mm, rotated rx 180 ry 0 rz -180 deg; joints [-14.167, -43.062, 107.778, 164.402, 65.537, -173.406]
  MoveL 233 to (240.65, 367.63, -2.5) mm, rotated rx -180 ry 0 rz 180 deg; joints [-14.224, -43.226, 108.27, 164.38, 65.859, -173.477]
  MoveL 234 to (233.21, 366.8, -2.5) mm, rotated rx 180 ry 0 rz -180 deg; joints [-14.263, -43.39, 108.765, 164.377, 66.182, -173.557]
  MoveL 235 to (225.83, 365.5, -2.5) mm, rotated rx 180 ry 0 rz 180 deg; joints [-14.284, -43.553, 109.262, 164.393, 66.506, -173.646]
  MoveL 236 to (218.56, 363.73, -2.5) mm, rotated rx -180 ry 0 rz -180 deg; joints [-14.288, -43.715, 109.759, 164.428, 66.829, -173.742]
  MoveL 237 to (211.41, 361.51, -2.5) mm, rotated rx -180 ry 0 rz -180 deg; joints [-14.273, -43.875, 110.253, 164.483, 67.149, -173.846]
  MoveL 238 to (204.41, 358.84, -2.5) mm, rotated rx 180 ry 0 rz -180 deg; joints [-14.239, -44.032, 110.743, 164.556, 67.467, -173.957]
  MoveL 239 to (197.6, 355.73, -2.5) mm, rotated rx -180 ry 0 rz -180 deg; joints [-14.186, -44.186, 111.228, 164.649, 67.78, -174.073]
  MoveL 240 to (191, 352.19, -2.5) mm, rotated rx -180 ry 0 rz -180 deg; joints [-14.114, -44.336, 111.704, 164.761, 68.087, -174.195]
  MoveL 241 to (184.64, 348.24, -2.5) mm, rotated rx 180 ry 0 rz 180 deg; joints [-14.023, -44.482, 112.17, 164.892, 68.387, -174.321]
  MoveL 242 to (178.54, 343.9, -2.5) mm, rotated rx -180 ry 0 rz 180 deg; joints [-13.913, -44.622, 112.624, 165.041, 68.679, -174.452]
  MoveL 243 to (172.73, 339.18, -2.5) mm, rotated rx 180 ry 0 rz 180 deg; joints [-13.785, -44.757, 113.064, 165.209, 68.962, -174.585]
  MoveL 244 to (167.23, 334.1, -2.5) mm, rotated rx 180 ry 0 rz -180 deg; joints [-13.639, -44.886, 113.488, 165.393, 69.234, -174.721]
  MoveL 245 to (162.06, 328.68, -2.5) mm, rotated rx -180 ry 0 rz 180 deg; joints [-13.474, -45.009, 113.895, 165.595, 69.494, -174.859]
  MoveL 246 to (157.25, 322.94, -2.5) mm, rotated rx -180 ry 0 rz -180 deg; joints [-13.292, -45.125, 114.283, 165.813, 69.742, -174.998]
  MoveL 247 to (152.81, 316.91, -2.5) mm, rotated rx 180 ry 0 rz 180 deg; joints [-13.094, -45.233, 114.65, 166.047, 69.975, -175.137]
  MoveL 248 to (148.76, 310.61, -2.5) mm, rotated rx -180 ry 0 rz 180 deg; joints [-12.879, -45.335, 114.994, 166.295, 70.193, -175.276]
  MoveL 249 to (145.12, 304.07, -2.5) mm, rotated rx 180 ry 0 rz -180 deg; joints [-12.65, -45.428, 115.315, 166.558, 70.395, -175.415]
  MoveL 250 to (141.9, 297.31, -2.5) mm, rotated rx -180 ry 0 rz 180 deg; joints [-12.406, -45.513, 115.609, 166.833, 70.58, -175.552]
  MoveL 251 to (139.12, 290.36, -2.5) mm, rotated rx -180 ry 0 rz 180 deg; joints [-12.149, -45.59, 115.878, 167.12, 70.746, -175.688]
  MoveL 252 to (136.78, 283.24, -2.5) mm, rotated rx 180 ry 0 rz 180 deg; joints [-11.879, -45.659, 116.118, 167.417, 70.894, -175.821]
  MoveL 253 to (134.9, 276, -2.5) mm, rotated rx 180 ry 0 rz 180 deg; joints [-11.6, -45.719, 116.329, 167.724, 71.021, -175.952]
  MoveL 254 to (133.48, 268.64, -2.5) mm, rotated rx 180 ry 0 rz 180 deg; joints [-11.31, -45.77, 116.511, 168.038, 71.129, -176.08]
  MoveL 255 to (132.53, 261.22, -2.5) mm, rotated rx 180 ry 0 rz 180 deg; joints [-11.013, -45.813, 116.661, 168.359, 71.214, -176.204]
  MoveL 256 to (132.06, 253.74, -2.5) mm, rotated rx -180 ry 0 rz -180 deg; joints [-10.709, -45.846, 116.78, 168.685, 71.279, -176.325]
  MoveL 257 to (132.06, 246.26, -2.5) mm, rotated rx -180 ry 0 rz -180 deg; joints [-10.4, -45.87, 116.867, 169.015, 71.321, -176.443]
  MoveL 258 to (132.53, 238.78, -2.5) mm, rotated rx -180 ry 0 rz 180 deg; joints [-10.087, -45.886, 116.922, 169.347, 71.34, -176.556]
  MoveL 259 to (133.48, 231.36, -2.5) mm, rotated rx 180 ry 0 rz 180 deg; joints [-9.773, -45.892, 116.944, 169.679, 71.337, -176.665]
  MoveL 260 to (134.9, 224, -2.5) mm, rotated rx 180 ry 0 rz -180 deg; joints [-9.458, -45.889, 116.933, 170.01, 71.312, -176.77]
  MoveL 261 to (136.78, 216.76, -2.5) mm, rotated rx -180 ry 0 rz 180 deg; joints [-9.145, -45.877, 116.89, 170.338, 71.264, -176.87]
  MoveL 262 to (139.12, 209.64, -2.5) mm, rotated rx -180 ry 0 rz 180 deg; joints [-8.835, -45.855, 116.814, 170.663, 71.193, -176.966]
  MoveL 263 to (141.9, 202.69, -2.5) mm, rotated rx -180 ry 0 rz -180 deg; joints [-8.529, -45.825, 116.706, 170.981, 71.1, -177.057]
  MoveL 264 to (145.12, 195.93, -2.5) mm, rotated rx 180 ry 0 rz -180 deg; joints [-8.229, -45.786, 116.566, 171.293, 70.986, -177.143]
  MoveL 265 to (148.76, 189.39, -2.5) mm, rotated rx -180 ry 0 rz -180 deg; joints [-7.937, -45.738, 116.395, 171.595, 70.85, -177.225]
  MoveL 266 to (152.81, 183.09, -2.5) mm, rotated rx 180 ry 0 rz -180 deg; joints [-7.653, -45.681, 116.194, 171.888, 70.694, -177.302]
  MoveL 267 to (157.25, 177.06, -2.5) mm, rotated rx 180 ry 0 rz 180 deg; joints [-7.38, -45.615, 115.964, 172.169, 70.518, -177.374]
  MoveL 268 to (162.06, 171.32, -2.5) mm, rotated rx -180 ry 0 rz 180 deg; joints [-7.119, -45.541, 115.705, 172.437, 70.323, -177.44]
  MoveL 269 to (167.23, 165.9, -2.5) mm, rotated rx 180 ry 0 rz 180 deg; joints [-6.87, -45.458, 115.419, 172.692, 70.111, -177.502]
  MoveL 270 to (172.73, 160.82, -2.5) mm, rotated rx 180 ry 0 rz -180 deg; joints [-6.636, -45.368, 115.108, 172.931, 69.881, -177.558]
  MoveL 271 to (178.54, 156.1, -2.5) mm, rotated rx -180 ry 0 rz -180 deg; joints [-6.416, -45.269, 114.771, 173.155, 69.636, -177.608]
  MoveL 272 to (184.64, 151.76, -2.5) mm, rotated rx 180 ry 0 rz 180 deg; joints [-6.212, -45.163, 114.412, 173.361, 69.376, -177.652]
  MoveL 273 to (191, 147.81, -2.5) mm, rotated rx -180 ry 0 rz 180 deg; joints [-6.024, -45.05, 114.031, 173.55, 69.103, -177.691]
  MoveL 274 to (197.6, 144.27, -2.5) mm, rotated rx 180 ry 0 rz 180 deg; joints [-5.853, -44.929, 113.631, 173.721, 68.818, -177.723]
  MoveL 275 to (204.41, 141.16, -2.5) mm, rotated rx 180 ry 0 rz -180 deg; joints [-5.701, -44.802, 113.212, 173.872, 68.522, -177.749]
  MoveL 276 to (211.41, 138.49, -2.5) mm, rotated rx -180 ry 0 rz -180 deg; joints [-5.566, -44.669, 112.777, 174.004, 68.216, -177.768]
  MoveL 277 to (218.56, 136.27, -2.5) mm, rotated rx 180 ry 0 rz 180 deg; joints [-5.45, -44.531, 112.328, 174.117, 67.903, -177.78]
  MoveL 278 to (225.83, 134.5, -2.5) mm, rotated rx -180 ry 0 rz 180 deg; joints [-5.353, -44.387, 111.866, 174.208, 67.582, -177.785]
  MoveL 279 to (233.21, 133.2, -2.5) mm, rotated rx -180 ry 0 rz 180 deg; joints [-5.274, -44.238, 111.393, 174.28, 67.257, -177.782]
  MoveL 280 to (240.65, 132.37, -2.5) mm, rotated rx 180 ry 0 rz 180 deg; joints [-5.215, -44.086, 110.911, 174.33, 66.927, -177.772]
  MoveL 281 to (248.13, 132.01, -2.5) mm, rotated rx -180 ry 0 rz 180 deg; joints [-5.174, -43.93, 110.423, 174.36, 66.595, -177.754]
  MoveL 282 to (255.61, 132.13, -2.5) mm, rotated rx 180 ry 0 rz 180 deg; joints [-5.153, -43.771, 109.93, 174.37, 66.261, -177.727]
  MoveL 283 to (263.08, 132.73, -2.5) mm, rotated rx 180 ry 0 rz 180 deg; joints [-5.15, -43.609, 109.433, 174.358, 65.928, -177.693]
  MoveL 284 to (270.49, 133.79, -2.5) mm, rotated rx 180 ry 0 rz 180 deg; joints [-5.165, -43.446, 108.936, 174.327, 65.596, -177.65]
  MoveL 285 to (277.82, 135.33, -2.5) mm, rotated rx -180 ry 0 rz -180 deg; joints [-5.198, -43.282, 108.44, 174.275, 65.267, -177.598]
  MoveL 286 to (285.04, 137.32, -2.5) mm, rotated rx 180 ry 0 rz -180 deg; joints [-5.249, -43.118, 107.948, 174.204, 64.942, -177.538]
  MoveL 287 to (292.11, 139.77, -2.5) mm, rotated rx -180 ry 0 rz -180 deg; joints [-5.317, -42.955, 107.46, 174.113, 64.622, -177.47]
  MoveL 288 to (299.02, 142.66, -2.5) mm, rotated rx -180 ry 0 rz -180 deg; joints [-5.402, -42.792, 106.979, 174.004, 64.309, -177.393]
  MoveL 289 to (305.73, 145.99, -2.5) mm, rotated rx -180 ry 0 rz -180 deg; joints [-5.503, -42.632, 106.506, 173.876, 64.004, -177.307]
  MoveL 290 to (312.21, 149.73, -2.5) mm, rotated rx -180 ry 0 rz -180 deg; joints [-5.619, -42.474, 106.045, 173.73, 63.708, -177.214]
  MoveL 291 to (318.45, 153.88, -2.5) mm, rotated rx 180 ry 0 rz 180 deg; joints [-5.75, -42.319, 105.595, 173.568, 63.421, -177.112]
  MoveL 292 to (324.41, 158.41, -2.5) mm, rotated rx 180 ry 0 rz 180 deg; joints [-5.896, -42.168, 105.16, 173.389, 63.146, -177.003]
  MoveL 293 to (330.06, 163.32, -2.5) mm, rotated rx 180 ry 0 rz -180 deg; joints [-6.055, -42.022, 104.741, 173.194, 62.883, -176.886]
  MoveL 294 to (335.4, 168.57, -2.5) mm, rotated rx 180 ry 0 rz 180 deg; joints [-6.226, -41.882, 104.338, 172.985, 62.633, -176.763]
  MoveL 295 to (340.39, 174.15, -2.5) mm, rotated rx -180 ry 0 rz -180 deg; joints [-6.41, -41.747, 103.955, 172.762, 62.397, -176.632]
  MoveL 296 to (345.02, 180.04, -2.5) mm, rotated rx 180 ry 0 rz -180 deg; joints [-6.605, -41.619, 103.593, 172.526, 62.176, -176.496]
  MoveL 297 to (349.27, 186.2, -2.5) mm, rotated rx 180 ry 0 rz 180 deg; joints [-6.811, -41.498, 103.252, 172.279, 61.971, -176.354]
  MoveL 298 to (353.11, 192.63, -2.5) mm, rotated rx -180 ry 0 rz -180 deg; joints [-7.027, -41.385, 102.934, 172.02, 61.782, -176.208]
  MoveL 299 to (356.55, 199.28, -2.5) mm, rotated rx 180 ry 0 rz -180 deg; joints [-7.251, -41.28, 102.64, 171.751, 61.611, -176.057]
  MoveL 300 to (359.55, 206.14, -2.5) mm, rotated rx -180 ry 0 rz 180 deg; joints [-7.484, -41.184, 102.372, 171.474, 61.457, -175.903]
  MoveL 301 to (362.11, 213.18, -2.5) mm, rotated rx -180 ry 0 rz 180 deg; joints [-7.724, -41.097, 102.131, 171.188, 61.321, -175.745]
  MoveL 302 to (364.22, 220.36, -2.5) mm, rotated rx -180 ry 0 rz 180 deg; joints [-7.97, -41.02, 101.917, 170.896, 61.205, -175.586]
  MoveL 303 to (365.87, 227.67, -2.5) mm, rotated rx -180 ry 0 rz -180 deg; joints [-8.222, -40.953, 101.731, 170.599, 61.107, -175.426]
  MoveL 304 to (367.05, 235.06, -2.5) mm, rotated rx 180 ry 0 rz 180 deg; joints [-8.479, -40.896, 101.574, 170.297, 61.029, -175.266]
  MoveL 305 to (367.76, 242.52, -2.5) mm, rotated rx 180 ry 0 rz -180 deg; joints [-8.74, -40.85, 101.447, 169.992, 60.971, -175.106]
  MoveL 306 to (368, 250, -2.5) mm, rotated rx -180 ry 0 rz -180 deg; joints [-9.004, -40.814, 101.349, 169.685, 60.933, -174.947]
  MoveL 307 to (356, 250, -2.5) mm, rotated rx 180 ry 0 rz 180 deg; joints [-9.072, -41.114, 102.177, 169.66, 61.459, -175.018]
  MoveL 308 to (355.79, 256.72, -2.5) mm, rotated rx -180 ry 0 rz -180 deg; joints [-9.313, -41.092, 102.117, 169.383, 61.443, -174.879]
  MoveL 309 to (355.15, 263.42, -2.5) mm, rotated rx 180 ry 0 rz -180 deg; joints [-9.555, -41.08, 102.085, 169.106, 61.444, -174.744]
  MoveL 310 to (354.08, 270.06, -2.5) mm, rotated rx -180 ry 0 rz 180 deg; joints [-9.798, -41.078, 102.08, 168.831, 61.464, -174.611]
  MoveL 311 to (352.6, 276.62, -2.5) mm, rotated rx -180 ry 0 rz -180 deg; joints [-10.041, -41.087, 102.103, 168.557, 61.501, -174.484]
  MoveL 312 to (350.71, 283.08, -2.5) mm, rotated rx -180 ry 0 rz 180 deg; joints [-10.282, -41.105, 102.153, 168.287, 61.556, -174.361]
  MoveL 313 to (348.41, 289.4, -2.5) mm, rotated rx 180 ry 0 rz -180 deg; joints [-10.522, -41.133, 102.231, 168.022, 61.629, -174.243]
  MoveL 314 to (345.71, 295.56, -2.5) mm, rotated rx -180 ry 0 rz 180 deg; joints [-10.759, -41.171, 102.337, 167.761, 61.719, -174.132]
  MoveL 315 to (342.63, 301.54, -2.5) mm, rotated rx 180 ry 0 rz 180 deg; joints [-10.993, -41.218, 102.469, 167.507, 61.826, -174.028]
  MoveL 316 to (339.17, 307.31, -2.5) mm, rotated rx -180 ry 0 rz -180 deg; joints [-11.222, -41.275, 102.627, 167.261, 61.949, -173.931]
  MoveL 317 to (335.36, 312.85, -2.5) mm, rotated rx 180 ry 0 rz -180 deg; joints [-11.447, -41.341, 102.811, 167.022, 62.088, -173.842]
  MoveL 318 to (331.2, 318.14, -2.5) mm, rotated rx 180 ry 0 rz -180 deg; joints [-11.665, -41.415, 103.02, 166.792, 62.242, -173.762]
  MoveL 319 to (326.72, 323.15, -2.5) mm, rotated rx 180 ry 0 rz 180 deg; joints [-11.878, -41.498, 103.253, 166.572, 62.412, -173.69]
  MoveL 320 to (321.92, 327.87, -2.5) mm, rotated rx -180 ry 0 rz 180 deg; joints [-12.083, -41.589, 103.509, 166.362, 62.595, -173.628]
  MoveL 321 to (316.84, 332.27, -2.5) mm, rotated rx 180 ry 0 rz -180 deg; joints [-12.28, -41.688, 103.788, 166.164, 62.792, -173.575]
  MoveL 322 to (311.49, 336.35, -2.5) mm, rotated rx 180 ry 0 rz 180 deg; joints [-12.468, -41.793, 104.087, 165.978, 63.001, -173.532]
  MoveL 323 to (305.89, 340.07, -2.5) mm, rotated rx 180 ry 0 rz -180 deg; joints [-12.647, -41.906, 104.407, 165.804, 63.223, -173.498]
  MoveL 324 to (300.06, 343.43, -2.5) mm, rotated rx 180 ry 0 rz 180 deg; joints [-12.815, -42.024, 104.745, 165.644, 63.455, -173.475]
  MoveL 325 to (294.03, 346.42, -2.5) mm, rotated rx 180 ry 0 rz 180 deg; joints [-12.973, -42.148, 105.101, 165.498, 63.698, -173.462]
  MoveL 326 to (287.83, 349.02, -2.5) mm, rotated rx -180 ry 0 rz 180 deg; joints [-13.119, -42.277, 105.473, 165.366, 63.95, -173.458]
  MoveL 327 to (281.47, 351.22, -2.5) mm, rotated rx 180 ry 0 rz 180 deg; joints [-13.253, -42.41, 105.86, 165.249, 64.21, -173.465]
  MoveL 328 to (274.99, 353.01, -2.5) mm, rotated rx 180 ry 0 rz 180 deg; joints [-13.375, -42.548, 106.26, 165.147, 64.478, -173.482]
  MoveL 329 to (268.41, 354.39, -2.5) mm, rotated rx 180 ry 0 rz 180 deg; joints [-13.483, -42.688, 106.672, 165.062, 64.752, -173.508]
  MoveL 330 to (261.75, 355.35, -2.5) mm, rotated rx -180 ry 0 rz -180 deg; joints [-13.577, -42.831, 107.093, 164.992, 65.031, -173.543]
  MoveL 331 to (255.04, 355.88, -2.5) mm, rotated rx -180 ry 0 rz -180 deg; joints [-13.656, -42.976, 107.523, 164.939, 65.316, -173.588]
  MoveL 332 to (248.32, 355.99, -2.5) mm, rotated rx 180 ry 0 rz -180 deg; joints [-13.721, -43.122, 107.96, 164.903, 65.603, -173.642]
  MoveL 333 to (241.6, 355.67, -2.5) mm, rotated rx 180 ry 0 rz -180 deg; joints [-13.77, -43.27, 108.402, 164.884, 65.893, -173.704]
  MoveL 334 to (234.91, 354.92, -2.5) mm, rotated rx -180 ry 0 rz -180 deg; joints [-13.803, -43.417, 108.847, 164.883, 66.184, -173.775]
  MoveL 335 to (228.29, 353.75, -2.5) mm, rotated rx -180 ry 0 rz 180 deg; joints [-13.821, -43.563, 109.293, 164.898, 66.475, -173.852]
  MoveL 336 to (221.75, 352.17, -2.5) mm, rotated rx 180 ry 0 rz 180 deg; joints [-13.821, -43.709, 109.739, 164.931, 66.766, -173.937]
  MoveL 337 to (215.33, 350.17, -2.5) mm, rotated rx -180 ry 0 rz 180 deg; joints [-13.806, -43.852, 110.183, 164.981, 67.054, -174.029]
  MoveL 338 to (209.05, 347.77, -2.5) mm, rotated rx 180 ry 0 rz 180 deg; joints [-13.773, -43.994, 110.624, 165.049, 67.34, -174.126]
  MoveL 339 to (202.93, 344.98, -2.5) mm, rotated rx -180 ry 0 rz -180 deg; joints [-13.723, -44.132, 111.058, 165.134, 67.621, -174.229]
  MoveL 340 to (197, 341.8, -2.5) mm, rotated rx 180 ry 0 rz 180 deg; joints [-13.657, -44.268, 111.486, 165.236, 67.897, -174.337]
  MoveL 341 to (191.28, 338.25, -2.5) mm, rotated rx -180 ry 0 rz -180 deg; joints [-13.574, -44.399, 111.904, 165.355, 68.166, -174.449]
  MoveL 342 to (185.81, 334.35, -2.5) mm, rotated rx 180 ry 0 rz -180 deg; joints [-13.474, -44.526, 112.311, 165.49, 68.428, -174.564]
  MoveL 343 to (180.58, 330.11, -2.5) mm, rotated rx -180 ry 0 rz -180 deg; joints [-13.357, -44.647, 112.706, 165.642, 68.681, -174.683]
  MoveL 344 to (175.64, 325.55, -2.5) mm, rotated rx 180 ry 0 rz 180 deg; joints [-13.224, -44.764, 113.086, 165.809, 68.925, -174.804]
  MoveL 345 to (171, 320.68, -2.5) mm, rotated rx 180 ry 0 rz -180 deg; joints [-13.076, -44.875, 113.451, 165.991, 69.158, -174.927]
  MoveL 346 to (166.68, 315.52, -2.5) mm, rotated rx -180 ry 0 rz 180 deg; joints [-12.912, -44.98, 113.799, 166.188, 69.379, -175.051]
  MoveL 347 to (162.69, 310.11, -2.5) mm, rotated rx -180 ry 0 rz -180 deg; joints [-12.733, -45.078, 114.127, 166.398, 69.588, -175.176]
  MoveL 348 to (159.05, 304.45, -2.5) mm, rotated rx -180 ry 0 rz -180 deg; joints [-12.54, -45.17, 114.436, 166.622, 69.782, -175.301]
  MoveL 349 to (155.78, 298.57, -2.5) mm, rotated rx 180 ry 0 rz -180 deg; joints [-12.334, -45.255, 114.723, 166.858, 69.962, -175.426]
  MoveL 350 to (152.89, 292.5, -2.5) mm, rotated rx 180 ry 0 rz -180 deg; joints [-12.115, -45.332, 114.987, 167.105, 70.127, -175.55]
  MoveL 351 to (150.39, 286.25, -2.5) mm, rotated rx 180 ry 0 rz 180 deg; joints [-11.885, -45.403, 115.227, 167.362, 70.275, -175.672]
  MoveL 352 to (148.29, 279.86, -2.5) mm, rotated rx 180 ry 0 rz 180 deg; joints [-11.645, -45.465, 115.442, 167.628, 70.406, -175.793]
  MoveL 353 to (146.6, 273.35, -2.5) mm, rotated rx 180 ry 0 rz -180 deg; joints [-11.395, -45.52, 115.631, 167.903, 70.519, -175.912]
  MoveL 354 to (145.33, 266.75, -2.5) mm, rotated rx -180 ry 0 rz -180 deg; joints [-11.137, -45.566, 115.793, 168.185, 70.614, -176.028]
  MoveL 355 to (144.48, 260.08, -2.5) mm, rotated rx 180 ry 0 rz -180 deg; joints [-10.872, -45.605, 115.928, 168.472, 70.69, -176.141]
  MoveL 356 to (144.05, 253.36, -2.5) mm, rotated rx -180 ry 0 rz 180 deg; joints [-10.601, -45.635, 116.034, 168.763, 70.747, -176.252]
  MoveL 357 to (144.05, 246.64, -2.5) mm, rotated rx -180 ry 0 rz 180 deg; joints [-10.325, -45.657, 116.112, 169.058, 70.784, -176.359]
  MoveL 358 to (144.48, 239.92, -2.5) mm, rotated rx 180 ry 0 rz -180 deg; joints [-10.047, -45.671, 116.161, 169.355, 70.801, -176.463]
  MoveL 359 to (145.33, 233.25, -2.5) mm, rotated rx -180 ry 0 rz 180 deg; joints [-9.767, -45.677, 116.181, 169.651, 70.798, -176.563]
  MoveL 360 to (146.6, 226.65, -2.5) mm, rotated rx 180 ry 0 rz 180 deg; joints [-9.487, -45.674, 116.171, 169.947, 70.774, -176.659]
  MoveL 361 to (148.29, 220.14, -2.5) mm, rotated rx 180 ry 0 rz -180 deg; joints [-9.208, -45.663, 116.132, 170.241, 70.731, -176.751]
  MoveL 362 to (150.39, 213.75, -2.5) mm, rotated rx 180 ry 0 rz 180 deg; joints [-8.931, -45.644, 116.065, 170.53, 70.668, -176.839]
  MoveL 363 to (152.89, 207.5, -2.5) mm, rotated rx -180 ry 0 rz 180 deg; joints [-8.659, -45.616, 115.968, 170.815, 70.585, -176.923]
  MoveL 364 to (155.78, 201.43, -2.5) mm, rotated rx 180 ry 0 rz -180 deg; joints [-8.391, -45.58, 115.843, 171.093, 70.482, -177.003]
  MoveL 365 to (159.05, 195.55, -2.5) mm, rotated rx -180 ry 0 rz 180 deg; joints [-8.131, -45.537, 115.69, 171.363, 70.361, -177.078]
  MoveL 366 to (162.69, 189.89, -2.5) mm, rotated rx -180 ry 0 rz 180 deg; joints [-7.878, -45.485, 115.51, 171.625, 70.222, -177.148]
  MoveL 367 to (166.68, 184.48, -2.5) mm, rotated rx -180 ry 0 rz -180 deg; joints [-7.634, -45.425, 115.304, 171.876, 70.065, -177.214]
  MoveL 368 to (171, 179.32, -2.5) mm, rotated rx 180 ry 0 rz 180 deg; joints [-7.4, -45.357, 115.072, 172.117, 69.891, -177.274]
  MoveL 369 to (175.64, 174.45, -2.5) mm, rotated rx -180 ry 0 rz -180 deg; joints [-7.177, -45.283, 114.816, 172.345, 69.701, -177.33]
  MoveL 370 to (180.58, 169.89, -2.5) mm, rotated rx 180 ry 0 rz -180 deg; joints [-6.967, -45.2, 114.537, 172.559, 69.497, -177.381]
  MoveL 371 to (185.81, 165.65, -2.5) mm, rotated rx 180 ry 0 rz -180 deg; joints [-6.769, -45.111, 114.236, 172.76, 69.278, -177.426]
  MoveL 372 to (191.28, 161.75, -2.5) mm, rotated rx 180 ry 0 rz -180 deg; joints [-6.586, -45.015, 113.914, 172.946, 69.046, -177.466]
  MoveL 373 to (197, 158.2, -2.5) mm, rotated rx 180 ry 0 rz 180 deg; joints [-6.417, -44.912, 113.573, 173.115, 68.801, -177.5]
  MoveL 374 to (202.93, 155.02, -2.5) mm, rotated rx -180 ry 0 rz -180 deg; joints [-6.263, -44.803, 113.214, 173.269, 68.546, -177.528]
  MoveL 375 to (209.05, 152.23, -2.5) mm, rotated rx 180 ry 0 rz 180 deg; joints [-6.124, -44.688, 112.839, 173.406, 68.282, -177.55]
  MoveL 376 to (215.33, 149.83, -2.5) mm, rotated rx 180 ry 0 rz 180 deg; joints [-6.002, -44.568, 112.449, 173.525, 68.008, -177.566]
  MoveL 377 to (221.75, 147.83, -2.5) mm, rotated rx -180 ry 0 rz 180 deg; joints [-5.896, -44.443, 112.046, 173.626, 67.727, -177.576]
  MoveL 378 to (228.29, 146.25, -2.5) mm, rotated rx 180 ry 0 rz 180 deg; joints [-5.807, -44.313, 111.631, 173.71, 67.441, -177.579]
  MoveL 379 to (234.91, 145.08, -2.5) mm, rotated rx 180 ry 0 rz 180 deg; joints [-5.735, -44.179, 111.207, 173.775, 67.149, -177.574]
  MoveL 380 to (241.6, 144.33, -2.5) mm, rotated rx -180 ry 0 rz -180 deg; joints [-5.679, -44.042, 110.774, 173.821, 66.853, -177.563]
  MoveL 381 to (248.32, 144.01, -2.5) mm, rotated rx -180 ry 0 rz 180 deg; joints [-5.641, -43.902, 110.336, 173.85, 66.555, -177.545]
  MoveL 382 to (255.04, 144.12, -2.5) mm, rotated rx 180 ry 0 rz 180 deg; joints [-5.619, -43.759, 109.893, 173.859, 66.256, -177.519]
  MoveL 383 to (261.75, 144.65, -2.5) mm, rotated rx -180 ry 0 rz -180 deg; joints [-5.615, -43.614, 109.447, 173.85, 65.957, -177.486]
  MoveL 384 to (268.41, 145.61, -2.5) mm, rotated rx -180 ry 0 rz -180 deg; joints [-5.626, -43.467, 109.001, 173.823, 65.659, -177.446]
  MoveL 385 to (274.99, 146.99, -2.5) mm, rotated rx -180 ry 0 rz -180 deg; joints [-5.654, -43.32, 108.555, 173.778, 65.363, -177.398]
  MoveL 386 to (281.47, 148.78, -2.5) mm, rotated rx -180 ry 0 rz -180 deg; joints [-5.698, -43.173, 108.112, 173.715, 65.071, -177.342]
  MoveL 387 to (287.83, 150.98, -2.5) mm, rotated rx 180 ry 0 rz 180 deg; joints [-5.757, -43.027, 107.673, 173.634, 64.784, -177.279]
  MoveL 388 to (294.03, 153.58, -2.5) mm, rotated rx -180 ry 0 rz -180 deg; joints [-5.831, -42.881, 107.241, 173.537, 64.502, -177.208]
  MoveL 389 to (300.06, 156.57, -2.5) mm, rotated rx 180 ry 0 rz -180 deg; joints [-5.921, -42.737, 106.816, 173.423, 64.227, -177.13]
  MoveL 390 to (305.89, 159.93, -2.5) mm, rotated rx 180 ry 0 rz 180 deg; joints [-6.024, -42.596, 106.401, 173.293, 63.961, -177.045]
  MoveL 391 to (311.49, 163.65, -2.5) mm, rotated rx 180 ry 0 rz -180 deg; joints [-6.14, -42.457, 105.997, 173.147, 63.703, -176.952]
  MoveL 392 to (316.84, 167.73, -2.5) mm, rotated rx 180 ry 0 rz 180 deg; joints [-6.27, -42.323, 105.605, 172.987, 63.455, -176.854]
  MoveL 393 to (321.92, 172.13, -2.5) mm, rotated rx 180 ry 0 rz -180 deg; joints [-6.412, -42.192, 105.228, 172.813, 63.218, -176.748]
  MoveL 394 to (326.72, 176.85, -2.5) mm, rotated rx -180 ry 0 rz -180 deg; joints [-6.566, -42.066, 104.866, 172.626, 62.993, -176.637]
  MoveL 395 to (331.2, 181.86, -2.5) mm, rotated rx 180 ry 0 rz 180 deg; joints [-6.731, -41.946, 104.522, 172.426, 62.781, -176.52]
  MoveL 396 to (335.36, 187.15, -2.5) mm, rotated rx -180 ry 0 rz -180 deg; joints [-6.907, -41.831, 104.195, 172.214, 62.582, -176.397]
  MoveL 397 to (339.17, 192.69, -2.5) mm, rotated rx 180 ry 0 rz 180 deg; joints [-7.092, -41.723, 103.889, 171.992, 62.397, -176.27]
  MoveL 398 to (342.63, 198.46, -2.5) mm, rotated rx -180 ry 0 rz -180 deg; joints [-7.286, -41.622, 103.603, 171.76, 62.226, -176.139]
  MoveL 399 to (345.71, 204.44, -2.5) mm, rotated rx 180 ry 0 rz 180 deg; joints [-7.488, -41.529, 103.339, 171.518, 62.072, -176.005]
  MoveL 400 to (348.41, 210.6, -2.5) mm, rotated rx -180 ry 0 rz 180 deg; joints [-7.698, -41.443, 103.098, 171.269, 61.933, -175.867]
  MoveL 401 to (350.71, 216.92, -2.5) mm, rotated rx 180 ry 0 rz -180 deg; joints [-7.914, -41.365, 102.88, 171.012, 61.811, -175.727]
  MoveL 402 to (352.6, 223.38, -2.5) mm, rotated rx -180 ry 0 rz -180 deg; joints [-8.137, -41.297, 102.688, 170.75, 61.705, -175.586]
  MoveL 403 to (354.08, 229.94, -2.5) mm, rotated rx 180 ry 0 rz 180 deg; joints [-8.365, -41.237, 102.52, 170.482, 61.617, -175.443]
  MoveL 404 to (355.15, 236.58, -2.5) mm, rotated rx 180 ry 0 rz -180 deg; joints [-8.597, -41.186, 102.379, 170.211, 61.547, -175.301]
  MoveL 405 to (355.79, 243.28, -2.5) mm, rotated rx 180 ry 0 rz 180 deg; joints [-8.833, -41.145, 102.265, 169.936, 61.494, -175.159]
  MoveL 406 to (356, 250, -2.5) mm, rotated rx 180 ry 0 rz 180 deg; joints [-9.072, -41.114, 102.177, 169.66, 61.459, -175.018]
  MoveL 407 to (344, 250, -2.5) mm, rotated rx -180 ry 0 rz 180 deg; joints [-9.141, -41.408, 103, 169.633, 61.985, -175.089]
  MoveL 408 to (343.81, 255.96, -2.5) mm, rotated rx -180 ry 0 rz 180 deg; joints [-9.356, -41.389, 102.947, 169.387, 61.97, -174.968]
  MoveL 409 to (343.24, 261.9, -2.5) mm, rotated rx -180 ry 0 rz -180 deg; joints [-9.573, -41.379, 102.918, 169.141, 61.971, -174.849]
  MoveL 410 to (342.3, 267.79, -2.5) mm, rotated rx 180 ry 0 rz 180 deg; joints [-9.79, -41.377, 102.914, 168.896, 61.988, -174.733]
  MoveL 411 to (340.99, 273.61, -2.5) mm, rotated rx 180 ry 0 rz -180 deg; joints [-10.006, -41.385, 102.934, 168.653, 62.021, -174.621]
  MoveL 412 to (339.31, 279.33, -2.5) mm, rotated rx 180 ry 0 rz 180 deg; joints [-10.222, -41.401, 102.979, 168.412, 62.069, -174.514]
  MoveL 413 to (337.27, 284.94, -2.5) mm, rotated rx -180 ry 0 rz -180 deg; joints [-10.436, -41.425, 103.048, 168.176, 62.134, -174.411]
  MoveL 414 to (334.88, 290.4, -2.5) mm, rotated rx 180 ry 0 rz 180 deg; joints [-10.648, -41.459, 103.142, 167.944, 62.213, -174.314]
  MoveL 415 to (332.14, 295.7, -2.5) mm, rotated rx 180 ry 0 rz -180 deg; joints [-10.857, -41.5, 103.259, 167.718, 62.308, -174.223]
  MoveL 416 to (329.08, 300.82, -2.5) mm, rotated rx 180 ry 0 rz 180 deg; joints [-11.061, -41.55, 103.4, 167.499, 62.417, -174.138]
  MoveL 417 to (325.7, 305.73, -2.5) mm, rotated rx 180 ry 0 rz -180 deg; joints [-11.262, -41.608, 103.563, 167.286, 62.541, -174.061]
  MoveL 418 to (322.01, 310.42, -2.5) mm, rotated rx 180 ry 0 rz 180 deg; joints [-11.457, -41.674, 103.749, 167.081, 62.678, -173.99]
  MoveL 419 to (318.03, 314.87, -2.5) mm, rotated rx -180 ry 0 rz -180 deg; joints [-11.646, -41.747, 103.956, 166.885, 62.829, -173.927]
  MoveL 420 to (313.78, 319.05, -2.5) mm, rotated rx -180 ry 0 rz 180 deg; joints [-11.828, -41.827, 104.183, 166.699, 62.992, -173.872]
  MoveL 421 to (309.27, 322.96, -2.5) mm, rotated rx -180 ry 0 rz -180 deg; joints [-12.003, -41.914, 104.431, 166.523, 63.167, -173.826]
  MoveL 422 to (304.53, 326.57, -2.5) mm, rotated rx 180 ry 0 rz 180 deg; joints [-12.17, -42.007, 104.697, 166.357, 63.353, -173.787]
  MoveL 423 to (299.56, 329.87, -2.5) mm, rotated rx 180 ry 0 rz 180 deg; joints [-12.329, -42.106, 104.981, 166.202, 63.55, -173.757]
  MoveL 424 to (294.39, 332.86, -2.5) mm, rotated rx -180 ry 0 rz -180 deg; joints [-12.478, -42.21, 105.281, 166.06, 63.756, -173.736]
  MoveL 425 to (289.05, 335.51, -2.5) mm, rotated rx -180 ry 0 rz 180 deg; joints [-12.618, -42.32, 105.597, 165.93, 63.972, -173.724]
  MoveL 426 to (283.55, 337.81, -2.5) mm, rotated rx -180 ry 0 rz -180 deg; joints [-12.747, -42.434, 105.928, 165.813, 64.196, -173.72]
  MoveL 427 to (277.91, 339.76, -2.5) mm, rotated rx -180 ry 0 rz -180 deg; joints [-12.865, -42.551, 106.271, 165.709, 64.428, -173.726]
  MoveL 428 to (272.16, 341.35, -2.5) mm, rotated rx -180 ry 0 rz -180 deg; joints [-12.972, -42.673, 106.626, 165.62, 64.666, -173.739]
  MoveL 429 to (266.32, 342.57, -2.5) mm, rotated rx -180 ry 0 rz -180 deg; joints [-13.067, -42.797, 106.992, 165.544, 64.91, -173.761]
  MoveL 430 to (260.42, 343.42, -2.5) mm, rotated rx -180 ry 0 rz -180 deg; joints [-13.149, -42.923, 107.366, 165.483, 65.159, -173.792]
  MoveL 431 to (254.47, 343.89, -2.5) mm, rotated rx 180 ry 0 rz -180 deg; joints [-13.218, -43.051, 107.747, 165.437, 65.412, -173.83]
  MoveL 432 to (248.51, 343.99, -2.5) mm, rotated rx 180 ry 0 rz 180 deg; joints [-13.273, -43.181, 108.135, 165.405, 65.667, -173.876]
  MoveL 433 to (242.55, 343.7, -2.5) mm, rotated rx -180 ry 0 rz -180 deg; joints [-13.315, -43.311, 108.527, 165.389, 65.925, -173.93]
  MoveL 434 to (236.62, 343.04, -2.5) mm, rotated rx -180 ry 0 rz -180 deg; joints [-13.343, -43.441, 108.922, 165.389, 66.184, -173.991]
  MoveL 435 to (230.75, 342.01, -2.5) mm, rotated rx -180 ry 0 rz 180 deg; joints [-13.356, -43.571, 109.318, 165.403, 66.443, -174.058]
  MoveL 436 to (224.95, 340.6, -2.5) mm, rotated rx -180 ry 0 rz -180 deg; joints [-13.355, -43.7, 109.713, 165.434, 66.701, -174.132]
  MoveL 437 to (219.26, 338.83, -2.5) mm, rotated rx -180 ry 0 rz -180 deg; joints [-13.339, -43.828, 110.107, 165.48, 66.957, -174.211]
  MoveL 438 to (213.68, 336.7, -2.5) mm, rotated rx 180 ry 0 rz 180 deg; joints [-13.309, -43.953, 110.497, 165.541, 67.21, -174.296]
  MoveL 439 to (208.26, 334.22, -2.5) mm, rotated rx 180 ry 0 rz 180 deg; joints [-13.263, -44.077, 110.883, 165.617, 67.459, -174.386]
  MoveL 440 to (203, 331.41, -2.5) mm, rotated rx -180 ry 0 rz 180 deg; joints [-13.202, -44.197, 111.261, 165.709, 67.704, -174.48]
  MoveL 441 to (197.93, 328.26, -2.5) mm, rotated rx -180 ry 0 rz -180 deg; joints [-13.127, -44.313, 111.632, 165.816, 67.942, -174.578]
  MoveL 442 to (193.07, 324.8, -2.5) mm, rotated rx 180 ry 0 rz 180 deg; joints [-13.037, -44.426, 111.992, 165.937, 68.174, -174.679]
  MoveL 443 to (188.44, 321.04, -2.5) mm, rotated rx -180 ry 0 rz 180 deg; joints [-12.932, -44.535, 112.342, 166.072, 68.398, -174.783]
  MoveL 444 to (184.06, 316.99, -2.5) mm, rotated rx -180 ry 0 rz -180 deg; joints [-12.813, -44.639, 112.679, 166.221, 68.614, -174.89]
  MoveL 445 to (179.95, 312.68, -2.5) mm, rotated rx -180 ry 0 rz -180 deg; joints [-12.681, -44.738, 113.002, 166.384, 68.819, -174.998]
  MoveL 446 to (176.11, 308.11, -2.5) mm, rotated rx -180 ry 0 rz 180 deg; joints [-12.535, -44.832, 113.309, 166.559, 69.015, -175.108]
  MoveL 447 to (172.57, 303.3, -2.5) mm, rotated rx -180 ry 0 rz 180 deg; joints [-12.376, -44.92, 113.6, 166.746, 69.198, -175.218]
  MoveL 448 to (169.35, 298.29, -2.5) mm, rotated rx -180 ry 0 rz -180 deg; joints [-12.205, -45.002, 113.872, 166.945, 69.37, -175.329]
  MoveL 449 to (166.45, 293.07, -2.5) mm, rotated rx 180 ry 0 rz 180 deg; joints [-12.022, -45.078, 114.126, 167.154, 69.529, -175.44]
  MoveL 450 to (163.89, 287.69, -2.5) mm, rotated rx -180 ry 0 rz -180 deg; joints [-11.829, -45.147, 114.359, 167.373, 69.673, -175.55]
  MoveL 451 to (161.67, 282.15, -2.5) mm, rotated rx 180 ry 0 rz -180 deg; joints [-11.626, -45.21, 114.572, 167.601, 69.803, -175.659]
  MoveL 452 to (159.81, 276.48, -2.5) mm, rotated rx -180 ry 0 rz -180 deg; joints [-11.414, -45.266, 114.762, 167.837, 69.918, -175.767]
  MoveL 453 to (158.31, 270.71, -2.5) mm, rotated rx 180 ry 0 rz 180 deg; joints [-11.193, -45.315, 114.929, 168.079, 70.018, -175.874]
  MoveL 454 to (157.18, 264.85, -2.5) mm, rotated rx 180 ry 0 rz 180 deg; joints [-10.966, -45.357, 115.072, 168.328, 70.101, -175.978]
  MoveL 455 to (156.43, 258.94, -2.5) mm, rotated rx -180 ry 0 rz 180 deg; joints [-10.733, -45.392, 115.191, 168.582, 70.167, -176.08]
  MoveL 456 to (156.05, 252.98, -2.5) mm, rotated rx -180 ry 0 rz 180 deg; joints [-10.494, -45.419, 115.285, 168.839, 70.217, -176.18]
  MoveL 457 to (156.05, 247.02, -2.5) mm, rotated rx 180 ry 0 rz -180 deg; joints [-10.252, -45.439, 115.354, 169.099, 70.249, -176.276]
  MoveL 458 to (156.43, 241.06, -2.5) mm, rotated rx -180 ry 0 rz 180 deg; joints [-10.007, -45.452, 115.397, 169.361, 70.263, -176.37]
  MoveL 459 to (157.18, 235.15, -2.5) mm, rotated rx 180 ry 0 rz 180 deg; joints [-9.761, -45.457, 115.414, 169.623, 70.26, -176.461]
  MoveL 460 to (158.31, 229.29, -2.5) mm, rotated rx -180 ry 0 rz -180 deg; joints [-9.515, -45.455, 115.406, 169.884, 70.239, -176.548]
  MoveL 461 to (159.81, 223.52, -2.5) mm, rotated rx 180 ry 0 rz 180 deg; joints [-9.27, -45.445, 115.372, 170.142, 70.2, -176.631]
  MoveL 462 to (161.67, 217.85, -2.5) mm, rotated rx -180 ry 0 rz 180 deg; joints [-9.026, -45.427, 115.312, 170.398, 70.144, -176.711]
  MoveL 463 to (163.89, 212.31, -2.5) mm, rotated rx 180 ry 0 rz -180 deg; joints [-8.787, -45.402, 115.226, 170.649, 70.071, -176.787]
  MoveL 464 to (166.45, 206.93, -2.5) mm, rotated rx 180 ry 0 rz 180 deg; joints [-8.551, -45.37, 115.116, 170.894, 69.981, -176.859]
  MoveL 465 to (169.35, 201.71, -2.5) mm, rotated rx 180 ry 0 rz 180 deg; joints [-8.322, -45.331, 114.981, 171.133, 69.874, -176.927]
  MoveL 466 to (172.57, 196.7, -2.5) mm, rotated rx -180 ry 0 rz 180 deg; joints [-8.099, -45.284, 114.822, 171.364, 69.751, -176.991]
  MoveL 467 to (176.11, 191.89, -2.5) mm, rotated rx -180 ry 0 rz 180 deg; joints [-7.884, -45.23, 114.64, 171.586, 69.613, -177.05]
  MoveL 468 to (179.95, 187.32, -2.5) mm, rotated rx 180 ry 0 rz 180 deg; joints [-7.677, -45.17, 114.435, 171.798, 69.46, -177.105]
  MoveL 469 to (184.06, 183.01, -2.5) mm, rotated rx 180 ry 0 rz -180 deg; joints [-7.48, -45.103, 114.209, 172, 69.292, -177.155]
  MoveL 470 to (188.44, 178.96, -2.5) mm, rotated rx 180 ry 0 rz -180 deg; joints [-7.294, -45.029, 113.962, 172.19, 69.112, -177.2]
  MoveL 471 to (193.07, 175.2, -2.5) mm, rotated rx -180 ry 0 rz 180 deg; joints [-7.119, -44.949, 113.696, 172.367, 68.919, -177.24]
  MoveL 472 to (197.93, 171.74, -2.5) mm, rotated rx -180 ry 0 rz -180 deg; joints [-6.956, -44.863, 113.411, 172.532, 68.714, -177.276]
  MoveL 473 to (203, 168.59, -2.5) mm, rotated rx -180 ry 0 rz 180 deg; joints [-6.806, -44.771, 113.109, 172.683, 68.499, -177.305]
  MoveL 474 to (208.26, 165.78, -2.5) mm, rotated rx -180 ry 0 rz 180 deg; joints [-6.668, -44.674, 112.792, 172.819, 68.274, -177.33]
  MoveL 475 to (213.68, 163.3, -2.5) mm, rotated rx 180 ry 0 rz 180 deg; joints [-6.545, -44.572, 112.46, 172.941, 68.04, -177.349]
  MoveL 476 to (219.26, 161.17, -2.5) mm, rotated rx -180 ry 0 rz -180 deg; joints [-6.435, -44.464, 112.114, 173.047, 67.798, -177.362]
  MoveL 477 to (224.95, 159.4, -2.5) mm, rotated rx 180 ry 0 rz 180 deg; joints [-6.34, -44.353, 111.757, 173.138, 67.55, -177.369]
  MoveL 478 to (230.75, 157.99, -2.5) mm, rotated rx -180 ry 0 rz -180 deg; joints [-6.259, -44.237, 111.39, 173.213, 67.296, -177.37]
  MoveL 479 to (236.62, 156.96, -2.5) mm, rotated rx 180 ry 0 rz 180 deg; joints [-6.194, -44.118, 111.014, 173.271, 67.038, -177.365]
  MoveL 480 to (242.55, 156.3, -2.5) mm, rotated rx -180 ry 0 rz -180 deg; joints [-6.143, -43.996, 110.631, 173.313, 66.777, -177.353]
  MoveL 481 to (248.51, 156.01, -2.5) mm, rotated rx -180 ry 0 rz -180 deg; joints [-6.107, -43.871, 110.242, 173.339, 66.513, -177.335]
  MoveL 482 to (254.47, 156.11, -2.5) mm, rotated rx 180 ry 0 rz 180 deg; joints [-6.086, -43.745, 109.849, 173.349, 66.248, -177.311]
  MoveL 483 to (260.42, 156.58, -2.5) mm, rotated rx -180 ry 0 rz -180 deg; joints [-6.08, -43.616, 109.454, 173.342, 65.983, -177.28]
  MoveL 484 to (266.32, 157.43, -2.5) mm, rotated rx -180 ry 0 rz -180 deg; joints [-6.088, -43.486, 109.058, 173.319, 65.719, -177.242]
  MoveL 485 to (272.16, 158.65, -2.5) mm, rotated rx 180 ry 0 rz 180 deg; joints [-6.111, -43.356, 108.663, 173.279, 65.456, -177.198]
  MoveL 486 to (277.91, 160.24, -2.5) mm, rotated rx 180 ry 0 rz -180 deg; joints [-6.148, -43.226, 108.27, 173.225, 65.197, -177.147]
  MoveL 487 to (283.55, 162.19, -2.5) mm, rotated rx 180 ry 0 rz 180 deg; joints [-6.199, -43.096, 107.881, 173.154, 64.942, -177.089]
  MoveL 488 to (289.05, 164.49, -2.5) mm, rotated rx 180 ry 0 rz 180 deg; joints [-6.263, -42.967, 107.497, 173.069, 64.692, -177.025]
  MoveL 489 to (294.39, 167.14, -2.5) mm, rotated rx 180 ry 0 rz -180 deg; joints [-6.341, -42.84, 107.12, 172.968, 64.449, -176.955]
  MoveL 490 to (299.56, 170.13, -2.5) mm, rotated rx 180 ry 0 rz -180 deg; joints [-6.431, -42.715, 106.751, 172.854, 64.212, -176.878]
  MoveL 491 to (304.53, 173.43, -2.5) mm, rotated rx 180 ry 0 rz -180 deg; joints [-6.534, -42.593, 106.393, 172.726, 63.983, -176.795]
  MoveL 492 to (309.27, 177.04, -2.5) mm, rotated rx 180 ry 0 rz 180 deg; joints [-6.648, -42.474, 106.045, 172.584, 63.762, -176.707]
  MoveL 493 to (313.78, 180.95, -2.5) mm, rotated rx -180 ry 0 rz -180 deg; joints [-6.773, -42.359, 105.71, 172.43, 63.552, -176.613]
  MoveL 494 to (318.03, 185.13, -2.5) mm, rotated rx 180 ry 0 rz 180 deg; joints [-6.909, -42.248, 105.389, 172.265, 63.352, -176.514]
  MoveL 495 to (322.01, 189.58, -2.5) mm, rotated rx -180 ry 0 rz -180 deg; joints [-7.056, -42.141, 105.083, 172.088, 63.163, -176.41]
  MoveL 496 to (325.7, 194.27, -2.5) mm, rotated rx 180 ry 0 rz -180 deg; joints [-7.211, -42.04, 104.793, 171.9, 62.985, -176.301]
  MoveL 497 to (329.08, 199.18, -2.5) mm, rotated rx -180 ry 0 rz -180 deg; joints [-7.375, -41.945, 104.52, 171.703, 62.821, -176.189]
  MoveL 498 to (332.14, 204.3, -2.5) mm, rotated rx -180 ry 0 rz 180 deg; joints [-7.548, -41.856, 104.266, 171.497, 62.669, -176.073]
  MoveL 499 to (334.88, 209.6, -2.5) mm, rotated rx 180 ry 0 rz 180 deg; joints [-7.728, -41.774, 104.032, 171.283, 62.531, -175.955]
  MoveL 500 to (337.27, 215.06, -2.5) mm, rotated rx -180 ry 0 rz -180 deg; joints [-7.915, -41.698, 103.818, 171.062, 62.408, -175.833]
  MoveL 501 to (339.31, 220.67, -2.5) mm, rotated rx -180 ry 0 rz -180 deg; joints [-8.108, -41.63, 103.625, 170.834, 62.299, -175.71]
  MoveL 502 to (340.99, 226.39, -2.5) mm, rotated rx 180 ry 0 rz 180 deg; joints [-8.306, -41.569, 103.454, 170.601, 62.205, -175.586]
  MoveL 503 to (342.3, 232.21, -2.5) mm, rotated rx -180 ry 0 rz 180 deg; joints [-8.509, -41.517, 103.305, 170.364, 62.126, -175.461]
  MoveL 504 to (343.24, 238.1, -2.5) mm, rotated rx 180 ry 0 rz 180 deg; joints [-8.717, -41.472, 103.18, 170.123, 62.063, -175.336]
  MoveL 505 to (343.81, 244.04, -2.5) mm, rotated rx 180 ry 0 rz 180 deg; joints [-8.928, -41.436, 103.078, 169.879, 62.016, -175.212]
  MoveL 506 to (344, 250, -2.5) mm, rotated rx -180 ry 0 rz 180 deg; joints [-9.141, -41.408, 103, 169.633, 61.985, -175.089]
  MoveL 507 to (332, 250, -2.5) mm, rotated rx -180 ry 0 rz -180 deg; joints [-9.211, -41.698, 103.818, 169.605, 62.51, -175.16]
  MoveL 508 to (331.83, 255.2, -2.5) mm, rotated rx 180 ry 0 rz 180 deg; joints [-9.4, -41.682, 103.771, 169.389, 62.496, -175.055]
  MoveL 509 to (331.34, 260.38, -2.5) mm, rotated rx 180 ry 0 rz -180 deg; joints [-9.59, -41.673, 103.746, 169.174, 62.497, -174.953]
  MoveL 510 to (330.52, 265.52, -2.5) mm, rotated rx -180 ry 0 rz -180 deg; joints [-9.781, -41.672, 103.742, 168.959, 62.511, -174.854]
  MoveL 511 to (329.37, 270.59, -2.5) mm, rotated rx -180 ry 0 rz 180 deg; joints [-9.972, -41.678, 103.76, 168.747, 62.54, -174.758]
  MoveL 512 to (327.91, 275.59, -2.5) mm, rotated rx -180 ry 0 rz 180 deg; joints [-10.161, -41.692, 103.8, 168.536, 62.582, -174.665]
  MoveL 513 to (326.13, 280.48, -2.5) mm, rotated rx -180 ry 0 rz -180 deg; joints [-10.349, -41.713, 103.86, 168.33, 62.638, -174.577]
  MoveL 514 to (324.04, 285.24, -2.5) mm, rotated rx 180 ry 0 rz 180 deg; joints [-10.535, -41.742, 103.942, 168.127, 62.708, -174.494]
  MoveL 515 to (321.66, 289.87, -2.5) mm, rotated rx -180 ry 0 rz 180 deg; joints [-10.719, -41.778, 104.044, 167.929, 62.791, -174.415]
  MoveL 516 to (318.98, 294.33, -2.5) mm, rotated rx -180 ry 0 rz 180 deg; joints [-10.898, -41.821, 104.167, 167.736, 62.886, -174.342]
  MoveL 517 to (316.03, 298.62, -2.5) mm, rotated rx -180 ry 0 rz 180 deg; joints [-11.074, -41.872, 104.31, 167.55, 62.994, -174.275]
  MoveL 518 to (312.82, 302.71, -2.5) mm, rotated rx -180 ry 0 rz 180 deg; joints [-11.245, -41.928, 104.472, 167.371, 63.114, -174.214]
  MoveL 519 to (309.35, 306.59, -2.5) mm, rotated rx -180 ry 0 rz 180 deg; joints [-11.411, -41.992, 104.653, 167.199, 63.245, -174.16]
  MoveL 520 to (305.64, 310.24, -2.5) mm, rotated rx 180 ry 0 rz -180 deg; joints [-11.57, -42.061, 104.852, 167.036, 63.388, -174.113]
  MoveL 521 to (301.71, 313.64, -2.5) mm, rotated rx 180 ry 0 rz 180 deg; joints [-11.724, -42.136, 105.068, 166.882, 63.541, -174.072]
  MoveL 522 to (297.56, 316.8, -2.5) mm, rotated rx 180 ry 0 rz -180 deg; joints [-11.87, -42.217, 105.301, 166.737, 63.704, -174.039]
  MoveL 523 to (293.23, 319.68, -2.5) mm, rotated rx -180 ry 0 rz -180 deg; joints [-12.008, -42.303, 105.549, 166.602, 63.876, -174.013]
  MoveL 524 to (288.73, 322.28, -2.5) mm, rotated rx -180 ry 0 rz -180 deg; joints [-12.138, -42.394, 105.812, 166.477, 64.057, -173.994]
  MoveL 525 to (284.06, 324.59, -2.5) mm, rotated rx 180 ry 0 rz 180 deg; joints [-12.26, -42.489, 106.088, 166.364, 64.246, -173.983]
  MoveL 526 to (279.26, 326.6, -2.5) mm, rotated rx -180 ry 0 rz 180 deg; joints [-12.372, -42.587, 106.376, 166.261, 64.442, -173.979]
  MoveL 527 to (274.35, 328.3, -2.5) mm, rotated rx 180 ry 0 rz -180 deg; joints [-12.474, -42.69, 106.676, 166.171, 64.645, -173.983]
  MoveL 528 to (269.33, 329.69, -2.5) mm, rotated rx 180 ry 0 rz 180 deg; joints [-12.566, -42.795, 106.986, 166.093, 64.853, -173.994]
  MoveL 529 to (264.24, 330.75, -2.5) mm, rotated rx 180 ry 0 rz -180 deg; joints [-12.648, -42.903, 107.306, 166.027, 65.067, -174.012]
  MoveL 530 to (259.09, 331.49, -2.5) mm, rotated rx -180 ry 0 rz -180 deg; joints [-12.718, -43.013, 107.632, 165.974, 65.285, -174.037]
  MoveL 531 to (253.9, 331.91, -2.5) mm, rotated rx -180 ry 0 rz -180 deg; joints [-12.777, -43.124, 107.965, 165.935, 65.506, -174.07]
  MoveL 532 to (248.7, 331.99, -2.5) mm, rotated rx 180 ry 0 rz -180 deg; joints [-12.824, -43.237, 108.304, 165.908, 65.729, -174.109]
  MoveL 533 to (243.5, 331.74, -2.5) mm, rotated rx 180 ry 0 rz -180 deg; joints [-12.859, -43.35, 108.646, 165.895, 65.955, -174.154]
  MoveL 534 to (238.33, 331.17, -2.5) mm, rotated rx -180 ry 0 rz -180 deg; joints [-12.882, -43.464, 108.99, 165.895, 66.181, -174.206]
  MoveL 535 to (233.21, 330.26, -2.5) mm, rotated rx 180 ry 0 rz -180 deg; joints [-12.892, -43.577, 109.336, 165.909, 66.407, -174.263]
  MoveL 536 to (228.15, 329.04, -2.5) mm, rotated rx -180 ry 0 rz -180 deg; joints [-12.89, -43.69, 109.681, 165.936, 66.633, -174.326]
  MoveL 537 to (223.18, 327.49, -2.5) mm, rotated rx 180 ry 0 rz -180 deg; joints [-12.874, -43.801, 110.024, 165.977, 66.856, -174.394]
  MoveL 538 to (218.32, 325.63, -2.5) mm, rotated rx 180 ry 0 rz 180 deg; joints [-12.846, -43.911, 110.365, 166.032, 67.077, -174.466]
  MoveL 539 to (213.59, 323.47, -2.5) mm, rotated rx 180 ry 0 rz 180 deg; joints [-12.804, -44.018, 110.7, 166.099, 67.295, -174.543]
  MoveL 540 to (209, 321.01, -2.5) mm, rotated rx -180 ry 0 rz -180 deg; joints [-12.75, -44.124, 111.03, 166.18, 67.508, -174.624]
  MoveL 541 to (204.58, 318.27, -2.5) mm, rotated rx -180 ry 0 rz 180 deg; joints [-12.683, -44.226, 111.353, 166.274, 67.716, -174.708]
  MoveL 542 to (200.34, 315.25, -2.5) mm, rotated rx 180 ry 0 rz -180 deg; joints [-12.603, -44.325, 111.667, 166.381, 67.918, -174.796]
  MoveL 543 to (196.3, 311.97, -2.5) mm, rotated rx -180 ry 0 rz -180 deg; joints [-12.51, -44.42, 111.972, 166.5, 68.113, -174.886]
  MoveL 544 to (192.48, 308.44, -2.5) mm, rotated rx -180 ry 0 rz 180 deg; joints [-12.406, -44.511, 112.265, 166.631, 68.3, -174.978]
  MoveL 545 to (188.89, 304.68, -2.5) mm, rotated rx 180 ry 0 rz 180 deg; joints [-12.29, -44.598, 112.546, 166.773, 68.479, -175.072]
  MoveL 546 to (185.54, 300.69, -2.5) mm, rotated rx 180 ry 0 rz 180 deg; joints [-12.162, -44.681, 112.814, 166.927, 68.648, -175.167]
  MoveL 547 to (182.46, 296.5, -2.5) mm, rotated rx 180 ry 0 rz 180 deg; joints [-12.023, -44.758, 113.067, 167.09, 68.808, -175.263]
  MoveL 548 to (179.65, 292.12, -2.5) mm, rotated rx -180 ry 0 rz -180 deg; joints [-11.874, -44.83, 113.304, 167.264, 68.956, -175.36]
  MoveL 549 to (177.12, 287.57, -2.5) mm, rotated rx 180 ry 0 rz 180 deg; joints [-11.715, -44.897, 113.525, 167.446, 69.094, -175.457]
  MoveL 550 to (174.88, 282.88, -2.5) mm, rotated rx -180 ry 0 rz -180 deg; joints [-11.547, -44.959, 113.728, 167.637, 69.219, -175.553]
  MoveL 551 to (172.95, 278.05, -2.5) mm, rotated rx 180 ry 0 rz 180 deg; joints [-11.37, -45.014, 113.912, 167.836, 69.332, -175.649]
  MoveL 552 to (171.32, 273.1, -2.5) mm, rotated rx -180 ry 0 rz 180 deg; joints [-11.186, -45.063, 114.077, 168.041, 69.431, -175.744]
  MoveL 553 to (170.01, 268.07, -2.5) mm, rotated rx 180 ry 0 rz -180 deg; joints [-10.995, -45.107, 114.223, 168.253, 69.517, -175.838]
  MoveL 554 to (169.03, 262.96, -2.5) mm, rotated rx -180 ry 0 rz -180 deg; joints [-10.798, -45.144, 114.347, 168.469, 69.588, -175.93]
  MoveL 555 to (168.37, 257.79, -2.5) mm, rotated rx 180 ry 0 rz -180 deg; joints [-10.596, -45.174, 114.45, 168.689, 69.645, -176.02]
  MoveL 556 to (168.04, 252.6, -2.5) mm, rotated rx -180 ry 0 rz 180 deg; joints [-10.389, -45.199, 114.532, 168.913, 69.687, -176.109]
  MoveL 557 to (168.04, 247.4, -2.5) mm, rotated rx -180 ry 0 rz 180 deg; joints [-10.18, -45.216, 114.592, 169.139, 69.715, -176.194]
  MoveL 558 to (168.37, 242.21, -2.5) mm, rotated rx -180 ry 0 rz -180 deg; joints [-9.968, -45.227, 114.629, 169.366, 69.727, -176.278]
  MoveL 559 to (169.03, 237.04, -2.5) mm, rotated rx -180 ry 0 rz 180 deg; joints [-9.755, -45.232, 114.645, 169.593, 69.724, -176.358]
  MoveL 560 to (170.01, 231.93, -2.5) mm, rotated rx 180 ry 0 rz 180 deg; joints [-9.542, -45.23, 114.637, 169.819, 69.705, -176.436]
  MoveL 561 to (171.32, 226.9, -2.5) mm, rotated rx -180 ry 0 rz -180 deg; joints [-9.33, -45.221, 114.607, 170.044, 69.671, -176.51]
  MoveL 562 to (172.95, 221.95, -2.5) mm, rotated rx -180 ry 0 rz -180 deg; joints [-9.12, -45.206, 114.555, 170.266, 69.623, -176.582]
  MoveL 563 to (174.88, 217.12, -2.5) mm, rotated rx -180 ry 0 rz -180 deg; joints [-8.912, -45.184, 114.481, 170.483, 69.559, -176.649]
  MoveL 564 to (177.12, 212.43, -2.5) mm, rotated rx -180 ry 0 rz -180 deg; joints [-8.709, -45.155, 114.385, 170.696, 69.48, -176.713]
  MoveL 565 to (179.65, 207.88, -2.5) mm, rotated rx -180 ry 0 rz 180 deg; joints [-8.51, -45.12, 114.268, 170.904, 69.388, -176.774]
  MoveL 566 to (182.46, 203.5, -2.5) mm, rotated rx -180 ry 0 rz -180 deg; joints [-8.316, -45.079, 114.13, 171.104, 69.281, -176.83]
  MoveL 567 to (185.54, 199.31, -2.5) mm, rotated rx -180 ry 0 rz 180 deg; joints [-8.13, -45.032, 113.971, 171.297, 69.161, -176.883]
  MoveL 568 to (188.89, 195.32, -2.5) mm, rotated rx -180 ry 0 rz 180 deg; joints [-7.95, -44.978, 113.793, 171.482, 69.028, -176.931]
  MoveL 569 to (192.48, 191.56, -2.5) mm, rotated rx -180 ry 0 rz -180 deg; joints [-7.779, -44.919, 113.597, 171.657, 68.883, -176.976]
  MoveL 570 to (196.3, 188.03, -2.5) mm, rotated rx 180 ry 0 rz -180 deg; joints [-7.617, -44.854, 113.382, 171.822, 68.727, -177.015]
  MoveL 571 to (200.34, 184.75, -2.5) mm, rotated rx 180 ry 0 rz -180 deg; joints [-7.465, -44.784, 113.151, 171.977, 68.559, -177.051]
  MoveL 572 to (204.58, 181.73, -2.5) mm, rotated rx 180 ry 0 rz 180 deg; joints [-7.322, -44.708, 112.903, 172.12, 68.382, -177.081]
  MoveL 573 to (209, 178.99, -2.5) mm, rotated rx -180 ry 0 rz -180 deg; joints [-7.191, -44.627, 112.64, 172.252, 68.195, -177.107]
  MoveL 574 to (213.59, 176.53, -2.5) mm, rotated rx -180 ry 0 rz -180 deg; joints [-7.07, -44.542, 112.364, 172.371, 67.999, -177.128]
  MoveL 575 to (218.32, 174.37, -2.5) mm, rotated rx -180 ry 0 rz 180 deg; joints [-6.962, -44.452, 112.074, 172.478, 67.796, -177.143]
  MoveL 576 to (223.18, 172.51, -2.5) mm, rotated rx 180 ry 0 rz -180 deg; joints [-6.865, -44.358, 111.774, 172.571, 67.586, -177.154]
  MoveL 577 to (228.15, 170.96, -2.5) mm, rotated rx 180 ry 0 rz 180 deg; joints [-6.781, -44.26, 111.463, 172.651, 67.371, -177.159]
  MoveL 578 to (233.21, 169.74, -2.5) mm, rotated rx -180 ry 0 rz -180 deg; joints [-6.709, -44.159, 111.143, 172.716, 67.15, -177.159]
  MoveL 579 to (238.33, 168.83, -2.5) mm, rotated rx -180 ry 0 rz -180 deg; joints [-6.65, -44.055, 110.815, 172.768, 66.926, -177.153]
  MoveL 580 to (243.5, 168.26, -2.5) mm, rotated rx 180 ry 0 rz -180 deg; joints [-6.605, -43.948, 110.481, 172.806, 66.698, -177.141]
  MoveL 581 to (248.7, 168.01, -2.5) mm, rotated rx 180 ry 0 rz 180 deg; joints [-6.572, -43.839, 110.142, 172.829, 66.468, -177.124]
  MoveL 582 to (253.9, 168.09, -2.5) mm, rotated rx -180 ry 0 rz 180 deg; joints [-6.552, -43.728, 109.8, 172.838, 66.237, -177.102]
  MoveL 583 to (259.09, 168.51, -2.5) mm, rotated rx 180 ry 0 rz -180 deg; joints [-6.545, -43.616, 109.455, 172.833, 66.006, -177.073]
  MoveL 584 to (264.24, 169.25, -2.5) mm, rotated rx 180 ry 0 rz -180 deg; joints [-6.55, -43.503, 109.109, 172.814, 65.776, -177.039]
  MoveL 585 to (269.33, 170.31, -2.5) mm, rotated rx 180 ry 0 rz -180 deg; joints [-6.569, -43.39, 108.765, 172.781, 65.547, -176.998]
  MoveL 586 to (274.35, 171.7, -2.5) mm, rotated rx -180 ry 0 rz 180 deg; joints [-6.6, -43.276, 108.422, 172.734, 65.321, -176.953]
  MoveL 587 to (279.26, 173.4, -2.5) mm, rotated rx 180 ry 0 rz 180 deg; joints [-6.643, -43.163, 108.082, 172.673, 65.098, -176.901]
  MoveL 588 to (284.06, 175.41, -2.5) mm, rotated rx -180 ry 0 rz -180 deg; joints [-6.697, -43.051, 107.747, 172.599, 64.88, -176.844]
  MoveL 589 to (288.73, 177.72, -2.5) mm, rotated rx -180 ry 0 rz 180 deg; joints [-6.764, -42.941, 107.418, 172.512, 64.667, -176.781]
  MoveL 590 to (293.23, 180.32, -2.5) mm, rotated rx 180 ry 0 rz 180 deg; joints [-6.842, -42.832, 107.096, 172.413, 64.46, -176.713]
  MoveL 591 to (297.56, 183.2, -2.5) mm, rotated rx 180 ry 0 rz -180 deg; joints [-6.93, -42.726, 106.782, 172.302, 64.26, -176.64]
  MoveL 592 to (301.71, 186.36, -2.5) mm, rotated rx 180 ry 0 rz 180 deg; joints [-7.029, -42.622, 106.479, 172.179, 64.068, -176.563]
  MoveL 593 to (305.64, 189.76, -2.5) mm, rotated rx 180 ry 0 rz -180 deg; joints [-7.138, -42.522, 106.186, 172.045, 63.883, -176.48]
  MoveL 594 to (309.35, 193.41, -2.5) mm, rotated rx -180 ry 0 rz -180 deg; joints [-7.256, -42.426, 105.905, 171.901, 63.708, -176.393]
  MoveL 595 to (312.82, 197.29, -2.5) mm, rotated rx -180 ry 0 rz -180 deg; joints [-7.383, -42.334, 105.638, 171.747, 63.543, -176.303]
  MoveL 596 to (316.03, 201.38, -2.5) mm, rotated rx 180 ry 0 rz -180 deg; joints [-7.519, -42.246, 105.385, 171.584, 63.388, -176.208]
  MoveL 597 to (318.98, 205.67, -2.5) mm, rotated rx -180 ry 0 rz -180 deg; joints [-7.663, -42.164, 105.147, 171.412, 63.244, -176.111]
  MoveL 598 to (321.66, 210.13, -2.5) mm, rotated rx 180 ry 0 rz 180 deg; joints [-7.813, -42.087, 104.925, 171.232, 63.111, -176.01]
  MoveL 599 to (324.04, 214.76, -2.5) mm, rotated rx -180 ry 0 rz -180 deg; joints [-7.971, -42.015, 104.72, 171.046, 62.99, -175.907]
  MoveL 600 to (326.13, 219.52, -2.5) mm, rotated rx 180 ry 0 rz 180 deg; joints [-8.134, -41.95, 104.533, 170.853, 62.882, -175.802]
  MoveL 601 to (327.91, 224.41, -2.5) mm, rotated rx -180 ry 0 rz 180 deg; joints [-8.304, -41.89, 104.364, 170.654, 62.786, -175.696]
  MoveL 602 to (329.37, 229.41, -2.5) mm, rotated rx 180 ry 0 rz 180 deg; joints [-8.478, -41.838, 104.214, 170.451, 62.704, -175.588]
  MoveL 603 to (330.52, 234.48, -2.5) mm, rotated rx 180 ry 0 rz 180 deg; joints [-8.656, -41.792, 104.085, 170.243, 62.635, -175.481]
  MoveL 604 to (331.34, 239.62, -2.5) mm, rotated rx 180 ry 0 rz 180 deg; joints [-8.838, -41.754, 103.975, 170.032, 62.579, -175.373]
  MoveL 605 to (331.83, 244.8, -2.5) mm, rotated rx -180 ry 0 rz -180 deg; joints [-9.023, -41.722, 103.886, 169.819, 62.537, -175.266]
  MoveL 606 to (332, 250, -2.5) mm, rotated rx -180 ry 0 rz -180 deg; joints [-9.211, -41.698, 103.818, 169.605, 62.51, -175.16]
  MoveL 607 to (320, 250, -2.5) mm, rotated rx 180 ry 0 rz -180 deg; joints [-9.282, -41.984, 104.631, 169.574, 63.035, -175.23]
  MoveL 608 to (319.86, 254.44, -2.5) mm, rotated rx 180 ry 0 rz -180 deg; joints [-9.445, -41.97, 104.592, 169.39, 63.023, -175.143]
  MoveL 609 to (319.44, 258.86, -2.5) mm, rotated rx 180 ry 0 rz -180 deg; joints [-9.608, -41.963, 104.57, 169.205, 63.023, -175.057]
  MoveL 610 to (318.74, 263.25, -2.5) mm, rotated rx -180 ry 0 rz -180 deg; joints [-9.772, -41.961, 104.567, 169.022, 63.035, -174.973]
  MoveL 611 to (317.76, 267.58, -2.5) mm, rotated rx -180 ry 0 rz 180 deg; joints [-9.936, -41.967, 104.582, 168.839, 63.059, -174.892]
  MoveL 612 to (316.5, 271.84, -2.5) mm, rotated rx -180 ry 0 rz 180 deg; joints [-10.099, -41.979, 104.616, 168.659, 63.096, -174.814]
  MoveL 613 to (314.99, 276.02, -2.5) mm, rotated rx -180 ry 0 rz -180 deg; joints [-10.261, -41.997, 104.667, 168.482, 63.143, -174.74]
  MoveL 614 to (313.2, 280.09, -2.5) mm, rotated rx -180 ry 0 rz -180 deg; joints [-10.421, -42.021, 104.737, 168.308, 63.203, -174.67]
  MoveL 615 to (311.17, 284.03, -2.5) mm, rotated rx 180 ry 0 rz 180 deg; joints [-10.579, -42.052, 104.825, 168.139, 63.273, -174.604]
  MoveL 616 to (308.89, 287.84, -2.5) mm, rotated rx 180 ry 0 rz -180 deg; joints [-10.733, -42.088, 104.93, 167.974, 63.355, -174.543]
  MoveL 617 to (306.37, 291.5, -2.5) mm, rotated rx -180 ry 0 rz 180 deg; joints [-10.884, -42.131, 105.052, 167.814, 63.447, -174.486]
  MoveL 618 to (303.62, 295, -2.5) mm, rotated rx -180 ry 0 rz -180 deg; joints [-11.03, -42.179, 105.191, 167.661, 63.55, -174.435]
  MoveL 619 to (300.66, 298.31, -2.5) mm, rotated rx -180 ry 0 rz -180 deg; joints [-11.172, -42.233, 105.346, 167.514, 63.662, -174.389]
  MoveL 620 to (297.5, 301.42, -2.5) mm, rotated rx 180 ry 0 rz -180 deg; joints [-11.309, -42.292, 105.516, 167.374, 63.784, -174.349]
  MoveL 621 to (294.14, 304.33, -2.5) mm, rotated rx -180 ry 0 rz -180 deg; joints [-11.44, -42.355, 105.701, 167.242, 63.915, -174.314]
  MoveL 622 to (290.6, 307.02, -2.5) mm, rotated rx -180 ry 0 rz -180 deg; joints [-11.565, -42.424, 105.9, 167.117, 64.055, -174.286]
  MoveL 623 to (286.91, 309.48, -2.5) mm, rotated rx 180 ry 0 rz -180 deg; joints [-11.683, -42.497, 106.112, 167.002, 64.202, -174.263]
  MoveL 624 to (283.06, 311.7, -2.5) mm, rotated rx -180 ry 0 rz -180 deg; joints [-11.794, -42.574, 106.336, 166.895, 64.357, -174.247]
  MoveL 625 to (279.08, 313.67, -2.5) mm, rotated rx -180 ry 0 rz -180 deg; joints [-11.898, -42.654, 106.572, 166.798, 64.519, -174.237]
  MoveL 626 to (274.98, 315.39, -2.5) mm, rotated rx 180 ry 0 rz 180 deg; joints [-11.993, -42.738, 106.819, 166.711, 64.687, -174.234]
  MoveL 627 to (270.78, 316.84, -2.5) mm, rotated rx -180 ry 0 rz -180 deg; joints [-12.08, -42.825, 107.076, 166.634, 64.861, -174.236]
  MoveL 628 to (266.5, 318.03, -2.5) mm, rotated rx -180 ry 0 rz 180 deg; joints [-12.158, -42.915, 107.341, 166.567, 65.039, -174.245]
  MoveL 629 to (262.16, 318.94, -2.5) mm, rotated rx -180 ry 0 rz -180 deg; joints [-12.226, -43.006, 107.613, 166.512, 65.222, -174.26]
  MoveL 630 to (257.76, 319.57, -2.5) mm, rotated rx 180 ry 0 rz -180 deg; joints [-12.285, -43.1, 107.893, 166.467, 65.409, -174.28]
  MoveL 631 to (253.33, 319.92, -2.5) mm, rotated rx -180 ry 0 rz -180 deg; joints [-12.335, -43.195, 108.177, 166.433, 65.598, -174.307]
  MoveL 632 to (248.89, 319.99, -2.5) mm, rotated rx -180 ry 0 rz -180 deg; joints [-12.374, -43.291, 108.466, 166.411, 65.789, -174.339]
  MoveL 633 to (244.45, 319.78, -2.5) mm, rotated rx 180 ry 0 rz -180 deg; joints [-12.402, -43.388, 108.758, 166.4, 65.982, -174.377]
  MoveL 634 to (240.04, 319.29, -2.5) mm, rotated rx 180 ry 0 rz 180 deg; joints [-12.42, -43.484, 109.052, 166.401, 66.176, -174.419]
  MoveL 635 to (235.66, 318.52, -2.5) mm, rotated rx 180 ry 0 rz -180 deg; joints [-12.428, -43.581, 109.347, 166.414, 66.369, -174.467]
  MoveL 636 to (231.35, 317.47, -2.5) mm, rotated rx -180 ry 0 rz -180 deg; joints [-12.424, -43.677, 109.642, 166.438, 66.562, -174.519]
  MoveL 637 to (227.11, 316.15, -2.5) mm, rotated rx 180 ry 0 rz -180 deg; joints [-12.409, -43.772, 109.935, 166.474, 66.753, -174.576]
  MoveL 638 to (222.96, 314.56, -2.5) mm, rotated rx -180 ry 0 rz -180 deg; joints [-12.384, -43.866, 110.226, 166.522, 66.942, -174.637]
  MoveL 639 to (218.92, 312.72, -2.5) mm, rotated rx 180 ry 0 rz 180 deg; joints [-12.347, -43.958, 110.512, 166.58, 67.127, -174.702]
  MoveL 640 to (215, 310.62, -2.5) mm, rotated rx 180 ry 0 rz 180 deg; joints [-12.299, -44.048, 110.793, 166.65, 67.309, -174.77]
  MoveL 641 to (211.23, 308.28, -2.5) mm, rotated rx -180 ry 0 rz 180 deg; joints [-12.241, -44.136, 111.069, 166.731, 67.487, -174.841]
  MoveL 642 to (207.61, 305.7, -2.5) mm, rotated rx -180 ry 0 rz -180 deg; joints [-12.172, -44.221, 111.337, 166.823, 67.659, -174.914]
  MoveL 643 to (204.16, 302.9, -2.5) mm, rotated rx 180 ry 0 rz 180 deg; joints [-12.092, -44.302, 111.596, 166.926, 67.825, -174.99]
  MoveL 644 to (200.9, 299.89, -2.5) mm, rotated rx 180 ry 0 rz -180 deg; joints [-12.002, -44.381, 111.846, 167.038, 67.984, -175.069]
  MoveL 645 to (197.83, 296.67, -2.5) mm, rotated rx -180 ry 0 rz -180 deg; joints [-11.902, -44.455, 112.085, 167.16, 68.136, -175.148]
  MoveL 646 to (194.98, 293.27, -2.5) mm, rotated rx -180 ry 0 rz -180 deg; joints [-11.793, -44.526, 112.313, 167.291, 68.28, -175.229]
  MoveL 647 to (192.34, 289.69, -2.5) mm, rotated rx 180 ry 0 rz -180 deg; joints [-11.674, -44.593, 112.529, 167.431, 68.415, -175.311]
  MoveL 648 to (189.94, 285.96, -2.5) mm, rotated rx -180 ry 0 rz -180 deg; joints [-11.547, -44.655, 112.731, 167.58, 68.542, -175.394]
  MoveL 649 to (187.78, 282.08, -2.5) mm, rotated rx 180 ry 0 rz -180 deg; joints [-11.412, -44.713, 112.919, 167.736, 68.658, -175.477]
  MoveL 650 to (185.87, 278.07, -2.5) mm, rotated rx -180 ry 0 rz -180 deg; joints [-11.269, -44.766, 113.091, 167.899, 68.764, -175.559]
  MoveL 651 to (184.22, 273.94, -2.5) mm, rotated rx 180 ry 0 rz 180 deg; joints [-11.118, -44.813, 113.248, 168.068, 68.859, -175.642]
  MoveL 652 to (182.84, 269.72, -2.5) mm, rotated rx 180 ry 0 rz 180 deg; joints [-10.962, -44.856, 113.389, 168.243, 68.943, -175.723]
  MoveL 653 to (181.72, 265.42, -2.5) mm, rotated rx -180 ry 0 rz 180 deg; joints [-10.8, -44.894, 113.512, 168.423, 69.016, -175.804]
  MoveL 654 to (180.88, 261.06, -2.5) mm, rotated rx -180 ry 0 rz -180 deg; joints [-10.633, -44.926, 113.618, 168.607, 69.076, -175.884]
  MoveL 655 to (180.32, 256.65, -2.5) mm, rotated rx 180 ry 0 rz 180 deg; joints [-10.461, -44.952, 113.706, 168.794, 69.124, -175.962]
  MoveL 656 to (180.04, 252.22, -2.5) mm, rotated rx 180 ry 0 rz -180 deg; joints [-10.287, -44.973, 113.776, 168.985, 69.159, -176.038]
  MoveL 657 to (180.04, 247.78, -2.5) mm, rotated rx 180 ry 0 rz -180 deg; joints [-10.109, -44.988, 113.827, 169.177, 69.182, -176.113]
  MoveL 658 to (180.32, 243.35, -2.5) mm, rotated rx 180 ry 0 rz 180 deg; joints [-9.93, -44.998, 113.858, 169.369, 69.192, -176.185]
  MoveL 659 to (180.88, 238.94, -2.5) mm, rotated rx 180 ry 0 rz 180 deg; joints [-9.75, -45.002, 113.871, 169.562, 69.189, -176.255]
  MoveL 660 to (181.72, 234.58, -2.5) mm, rotated rx 180 ry 0 rz 180 deg; joints [-9.569, -45, 113.865, 169.755, 69.173, -176.323]
  MoveL 661 to (182.84, 230.28, -2.5) mm, rotated rx 180 ry 0 rz 180 deg; joints [-9.39, -44.992, 113.84, 169.945, 69.144, -176.388]
  MoveL 662 to (184.22, 226.06, -2.5) mm, rotated rx 180 ry 0 rz 180 deg; joints [-9.212, -44.979, 113.795, 170.133, 69.103, -176.45]
  MoveL 663 to (185.87, 221.93, -2.5) mm, rotated rx -180 ry 0 rz -180 deg; joints [-9.036, -44.96, 113.732, 170.318, 69.048, -176.509]
  MoveL 664 to (187.78, 217.92, -2.5) mm, rotated rx 180 ry 0 rz -180 deg; joints [-8.863, -44.935, 113.651, 170.499, 68.982, -176.565]
  MoveL 665 to (189.94, 214.04, -2.5) mm, rotated rx -180 ry 0 rz 180 deg; joints [-8.695, -44.905, 113.551, 170.675, 68.903, -176.618]
  MoveL 666 to (192.34, 210.31, -2.5) mm, rotated rx 180 ry 0 rz 180 deg; joints [-8.531, -44.87, 113.433, 170.846, 68.812, -176.667]
  MoveL 667 to (194.98, 206.73, -2.5) mm, rotated rx -180 ry 0 rz 180 deg; joints [-8.372, -44.829, 113.299, 171.01, 68.711, -176.712]
  MoveL 668 to (197.83, 203.33, -2.5) mm, rotated rx 180 ry 0 rz 180 deg; joints [-8.22, -44.783, 113.147, 171.167, 68.598, -176.754]
  MoveL 669 to (200.9, 200.11, -2.5) mm, rotated rx -180 ry 0 rz 180 deg; joints [-8.074, -44.732, 112.98, 171.316, 68.475, -176.792]
  MoveL 670 to (204.16, 197.1, -2.5) mm, rotated rx 180 ry 0 rz -180 deg; joints [-7.936, -44.676, 112.797, 171.457, 68.342, -176.827]
  MoveL 671 to (207.61, 194.3, -2.5) mm, rotated rx -180 ry 0 rz 180 deg; joints [-7.806, -44.615, 112.6, 171.589, 68.2, -176.857]
  MoveL 672 to (211.23, 191.72, -2.5) mm, rotated rx -180 ry 0 rz 180 deg; joints [-7.684, -44.55, 112.389, 171.711, 68.049, -176.883]
  MoveL 673 to (215, 189.38, -2.5) mm, rotated rx 180 ry 0 rz -180 deg; joints [-7.572, -44.48, 112.165, 171.823, 67.89, -176.904]
  MoveL 674 to (218.92, 187.28, -2.5) mm, rotated rx -180 ry 0 rz 180 deg; joints [-7.468, -44.407, 111.93, 171.925, 67.724, -176.922]
  MoveL 675 to (222.96, 185.44, -2.5) mm, rotated rx -180 ry 0 rz -180 deg; joints [-7.375, -44.33, 111.683, 172.016, 67.551, -176.934]
  MoveL 676 to (227.11, 183.85, -2.5) mm, rotated rx -180 ry 0 rz -180 deg; joints [-7.292, -44.249, 111.427, 172.096, 67.373, -176.943]
  MoveL 677 to (231.35, 182.53, -2.5) mm, rotated rx 180 ry 0 rz -180 deg; joints [-7.219, -44.165, 111.162, 172.165, 67.189, -176.946]
  MoveL 678 to (235.66, 181.48, -2.5) mm, rotated rx -180 ry 0 rz 180 deg; joints [-7.157, -44.079, 110.889, 172.222, 67.002, -176.945]
  MoveL 679 to (240.04, 180.71, -2.5) mm, rotated rx 180 ry 0 rz 180 deg; joints [-7.105, -43.989, 110.61, 172.266, 66.81, -176.939]
  MoveL 680 to (244.45, 180.22, -2.5) mm, rotated rx -180 ry 0 rz -180 deg; joints [-7.065, -43.898, 110.325, 172.299, 66.617, -176.928]
  MoveL 681 to (248.89, 180.01, -2.5) mm, rotated rx 180 ry 0 rz 180 deg; joints [-7.035, -43.805, 110.036, 172.32, 66.421, -176.912]
  MoveL 682 to (253.33, 180.08, -2.5) mm, rotated rx -180 ry 0 rz -180 deg; joints [-7.017, -43.71, 109.743, 172.328, 66.224, -176.892]
  MoveL 683 to (257.76, 180.43, -2.5) mm, rotated rx 180 ry 0 rz 180 deg; joints [-7.01, -43.614, 109.449, 172.325, 66.027, -176.866]
  MoveL 684 to (262.16, 181.06, -2.5) mm, rotated rx -180 ry 0 rz -180 deg; joints [-7.013, -43.518, 109.154, 172.309, 65.83, -176.835]
  MoveL 685 to (266.5, 181.97, -2.5) mm, rotated rx 180 ry 0 rz -180 deg; joints [-7.027, -43.421, 108.86, 172.281, 65.635, -176.8]
  MoveL 686 to (270.78, 183.16, -2.5) mm, rotated rx -180 ry 0 rz -180 deg; joints [-7.052, -43.324, 108.567, 172.242, 65.442, -176.759]
  MoveL 687 to (274.98, 184.61, -2.5) mm, rotated rx 180 ry 0 rz 180 deg; joints [-7.088, -43.228, 108.277, 172.191, 65.252, -176.714]
  MoveL 688 to (279.08, 186.33, -2.5) mm, rotated rx 180 ry 0 rz -180 deg; joints [-7.134, -43.133, 107.99, 172.129, 65.066, -176.664]
  MoveL 689 to (283.06, 188.3, -2.5) mm, rotated rx -180 ry 0 rz -180 deg; joints [-7.189, -43.039, 107.709, 172.055, 64.884, -176.61]
  MoveL 690 to (286.91, 190.52, -2.5) mm, rotated rx -180 ry 0 rz -180 deg; joints [-7.255, -42.946, 107.434, 171.971, 64.707, -176.551]
  MoveL 691 to (290.6, 192.98, -2.5) mm, rotated rx 180 ry 0 rz 180 deg; joints [-7.33, -42.856, 107.166, 171.877, 64.535, -176.488]
  MoveL 692 to (294.14, 195.67, -2.5) mm, rotated rx 180 ry 0 rz 180 deg; joints [-7.413, -42.768, 106.907, 171.772, 64.371, -176.421]
  MoveL 693 to (297.5, 198.58, -2.5) mm, rotated rx 180 ry 0 rz 180 deg; joints [-7.506, -42.683, 106.657, 171.659, 64.213, -176.35]
  MoveL 694 to (300.66, 201.69, -2.5) mm, rotated rx 180 ry 0 rz -180 deg; joints [-7.606, -42.601, 106.417, 171.536, 64.063, -176.276]
  MoveL 695 to (303.62, 205, -2.5) mm, rotated rx -180 ry 0 rz -180 deg; joints [-7.715, -42.523, 106.188, 171.405, 63.921, -176.198]
  MoveL 696 to (306.37, 208.5, -2.5) mm, rotated rx -180 ry 0 rz -180 deg; joints [-7.83, -42.449, 105.971, 171.265, 63.789, -176.118]
  MoveL 697 to (308.89, 212.16, -2.5) mm, rotated rx 180 ry 0 rz -180 deg; joints [-7.953, -42.379, 105.768, 171.119, 63.665, -176.035]
  MoveL 698 to (311.17, 215.97, -2.5) mm, rotated rx -180 ry 0 rz -180 deg; joints [-8.082, -42.313, 105.578, 170.966, 63.551, -175.949]
  MoveL 699 to (313.2, 219.91, -2.5) mm, rotated rx 180 ry 0 rz 180 deg; joints [-8.217, -42.252, 105.403, 170.806, 63.448, -175.862]
  MoveL 700 to (314.99, 223.98, -2.5) mm, rotated rx 180 ry 0 rz 180 deg; joints [-8.357, -42.197, 105.243, 170.641, 63.355, -175.773]
  MoveL 701 to (316.51, 228.16, -2.5) mm, rotated rx 180 ry 0 rz -180 deg; joints [-8.502, -42.147, 105.098, 170.472, 63.273, -175.683]
  MoveL 702 to (317.76, 232.42, -2.5) mm, rotated rx 180 ry 0 rz -180 deg; joints [-8.652, -42.102, 104.97, 170.298, 63.202, -175.592]
  MoveL 703 to (318.73, 236.75, -2.5) mm, rotated rx -180 ry 0 rz -180 deg; joints [-8.805, -42.064, 104.859, 170.12, 63.142, -175.501]
  MoveL 704 to (319.44, 241.14, -2.5) mm, rotated rx 180 ry 0 rz 180 deg; joints [-8.962, -42.031, 104.766, 169.94, 63.095, -175.41]
  MoveL 705 to (319.86, 245.56, -2.5) mm, rotated rx 180 ry 0 rz -180 deg; joints [-9.121, -42.004, 104.69, 169.758, 63.059, -175.32]
  MoveL 706 to (320, 250, -2.5) mm, rotated rx 180 ry 0 rz -180 deg; joints [-9.282, -41.984, 104.631, 169.574, 63.035, -175.23]
  MoveL 707 to (308, 250, -2.5) mm, rotated rx -180 ry 0 rz -180 deg; joints [-9.354, -42.265, 105.44, 169.542, 63.559, -175.301]
  MoveL 708 to (307.88, 253.68, -2.5) mm, rotated rx 180 ry 0 rz 180 deg; joints [-9.49, -42.254, 105.407, 169.388, 63.549, -175.23]
  MoveL 709 to (307.53, 257.34, -2.5) mm, rotated rx -180 ry 0 rz -180 deg; joints [-9.626, -42.248, 105.389, 169.235, 63.549, -175.159]
  MoveL 710 to (306.95, 260.98, -2.5) mm, rotated rx -180 ry 0 rz -180 deg; joints [-9.764, -42.247, 105.386, 169.083, 63.559, -175.091]
  MoveL 711 to (306.14, 264.57, -2.5) mm, rotated rx -180 ry 0 rz -180 deg; joints [-9.9, -42.251, 105.399, 168.931, 63.579, -175.025]
  MoveL 712 to (305.1, 268.1, -2.5) mm, rotated rx 180 ry 0 rz 180 deg; joints [-10.037, -42.261, 105.427, 168.781, 63.609, -174.962]
  MoveL 713 to (303.85, 271.56, -2.5) mm, rotated rx 180 ry 0 rz -180 deg; joints [-10.172, -42.276, 105.47, 168.634, 63.648, -174.901]
  MoveL 714 to (302.37, 274.93, -2.5) mm, rotated rx -180 ry 0 rz -180 deg; joints [-10.305, -42.296, 105.528, 168.489, 63.698, -174.844]
  MoveL 715 to (300.68, 278.2, -2.5) mm, rotated rx 180 ry 0 rz -180 deg; joints [-10.436, -42.321, 105.601, 168.348, 63.756, -174.79]
  MoveL 716 to (298.79, 281.36, -2.5) mm, rotated rx 180 ry 0 rz 180 deg; joints [-10.565, -42.351, 105.688, 168.211, 63.824, -174.74]
  MoveL 717 to (296.71, 284.39, -2.5) mm, rotated rx -180 ry 0 rz 180 deg; joints [-10.691, -42.386, 105.79, 168.078, 63.9, -174.693]
  MoveL 718 to (294.43, 287.28, -2.5) mm, rotated rx -180 ry 0 rz -180 deg; joints [-10.813, -42.426, 105.905, 167.951, 63.986, -174.651]
  MoveL 719 to (291.98, 290.02, -2.5) mm, rotated rx -180 ry 0 rz -180 deg; joints [-10.931, -42.47, 106.033, 167.828, 64.079, -174.614]
  MoveL 720 to (289.35, 292.61, -2.5) mm, rotated rx 180 ry 0 rz -180 deg; joints [-11.045, -42.518, 106.175, 167.712, 64.181, -174.581]
